(* PLC project TC3_TE1400_GeneratedModule_ModelBROSMattia_FB, Beckhoff Automation GmbH & Co. KG TwinCAT 3 Function - TE1400 1.2.1228 *)
(* stored: companyURL www.beckhoff.com, creationDateTime 2017-06-19T08:04:46 *)

TYPE E_TcMatSimDataAreaType : (NotSpecified := 0, Standard, InputSrc, InputDst, OutputSrc, OutputDst, InternalDa, MArea, RetainDa);
END_TYPE

TYPE ST_TcMatSimObjectDataAreaInfo : STRUCT
  pPlcVar : PVOID;
  pModuleProcImg : PVOID;
  nSize : UDINT;
  nDataAreaId : UDINT;
  eDataAreaType : E_TcMatSimDataAreaType;
END_STRUCT;
END_TYPE

{attribute 'pack_mode' := '4'}
TYPE ST_ModelBROSMattia_InitData : STRUCT
  Header : TComInitDataHdr;
  CallByHdr : TComInitDataElmHdr;
  CallBy : TctModuleCallByType;
  ExecutionSequenceHdr : TComInitDataElmHdr;
  ExecutionSequence : TctModuleExecutionSequenceType;
  StepSizeHdr : TComInitDataElmHdr;
  StepSize : TctStepSizeType;
  ExtendedFileAccessOIDHdr : TComInitDataElmHdr;
  ExtendedFileAccessOID : OTCID;
  ExtModeParametersHdr : TComInitDataElmHdr;
  ExtModeParameters : TctExtModeParametersType;
  ExecuteModelCodeHdr : TComInitDataElmHdr;
  ExecuteModelCode : BOOL;
  ModelParametersHdr : TComInitDataElmHdr;
  ModelParameters : P_model_bros_mattia_T;
  ContextInfoArr_0_TaskOidHdr : TComInitDataElmHdr;
  ContextInfoArr_0_TaskOid : OTCID;
  ContextInfoArr_0_TaskPriorityHdr : TComInitDataElmHdr;
  ContextInfoArr_0_TaskPriority : UDINT;
  ContextInfoArr_0_TaskCycleTimeNsHdr : TComInitDataElmHdr;
  ContextInfoArr_0_TaskCycleTimeNs : UDINT;
  ContextInfoArr_0_TaskPortHdr : TComInitDataElmHdr;
  ContextInfoArr_0_TaskPort : UINT;
  ContextInfoArr_0_TaskSortOrderHdr : TComInitDataElmHdr;
  ContextInfoArr_0_TaskSortOrder : UDINT;
END_STRUCT;
END_TYPE

TYPE ST_ModelBROSMattia_Input : STRUCT
  StatusWord_joint1 : UINT;
  MotorEncoder_joint1 : DINT;
  JointAbsEnc_joint1 : DINT;
  MotorCurrentAct_joint1 : INT;
  StatusWord_joint2 : UINT;
  MotorEncoder_joint2 : DINT;
  JointAbsEnc_joint2 : DINT;
  MotorCurrentAct_joint2 : INT;
  FTch1 : REAL;
  FTch2 : REAL;
  FTch3 : REAL;
  FTch4 : REAL;
  FTch5 : REAL;
  FTch6 : REAL;
  StatusWord_joint3 : UINT;
  MotorEncoder_joint3 : DINT;
  JointAbsEnc_joint3 : DINT;
  MotorCurrentAct_joint3 : INT;
  StatusWord_joint4 : UINT;
  MotorEncoder_joint4 : DINT;
  JointAbsEnc_joint4 : DINT;
  MotorCurrentAct_joint4 : INT;
  FTch7 : REAL;
  FTch8 : REAL;
  FTch9 : REAL;
  FTch10 : REAL;
  FTch11 : REAL;
  FTch12 : REAL;
END_STRUCT;
END_TYPE

TYPE ST_ModelBROSMattia_Output : STRUCT
  EnableCircuit1 : BOOL;
  ControlWord_joint1 : UINT;
  ModesOfOperation_joint1 : SINT;
  TargetCurrent_joint1 : INT;
  ControlWord_joint2 : UINT;
  ModesOfOperation_joint2 : SINT;
  TargetCurrent_joint2 : INT;
  EnableCircuit2 : BOOL;
  ControlWord_joint3 : UINT;
  ModesOfOperation_joint3 : SINT;
  TargetCurrent_joint3 : INT;
  ControlWord_joint4 : UINT;
  ModesOfOperation_joint4 : SINT;
  TargetCurrent_joint4 : INT;
  pause_logger : BOOL;
  DataToADS : matrix_9_real_T;
END_STRUCT;
END_TYPE

FUNCTION_BLOCK FB_TcMatSimObject
  VAR_INPUT
    bWriteFbInputValues : BOOL := TRUE;  (* set this flag to write FB input values to the TcComObject's input DataAreas. This will overwrite the mapped input values before module execution. Set to FALSE to read the mapped input values from the TcComObject to the FB. *)
  END_VAR
  VAR
    pDataAreas : POINTER TO ST_TcMatSimObjectDataAreaInfo;  (* process image src and dst pointers and sizes *)
    nDataAreas : UDINT;
    ipObjSrv : ITComObjectServer;  (* global interface pointers *)
    ipTcComObj : ITComObject;  (* object interface pointers *)
    ipTcCyclic : ITcCyclic;
    ipTcPostCyclic : ITcPostCyclic;
    ipTcAdi : ITcADI;
    ipTask : ITcTask;  (* task interface pointers *)
    pInitData : POINTER TO TComInitDataHdr;  (* initial parameters *)
    hResult : HRESULT;  (* hResult of interface calls (0 if no error) *)
    moduleClsId : CLSID;  (* module class ID *)
    assignedClsId : CLSID;  (* expected/desired module class ID *)
    bClassIdVerified : BOOL;
    bDynInstance : BOOL;  (* flag indicating whether the module instance was created dynamically *)
    eInitialObjState : TCOM_STATE := TCOM_STATE.TCOM_STATE_INIT;  (* the object state at the time FB_init was called, FB_exit will try to switch to this state (only if this means to shift down) *)
  END_VAR

            
          

{attribute 'object_name' := 'ReleaseTcComInterface'}
METHOD ReleaseTcComInterface : HRESULT
  VAR
    nStateChangeCnt : DINT := 0;
  END_VAR
                  
IF (ipTcComObj<>0) THEN
  WHILE (State>eInitialObjState AND nStateChangeCnt<1000) DO
    State := eInitialObjState;
    nStateChangeCnt := nStateChangeCnt+1;
  END_WHILE
  ReleaseObjInterfaces();
  IF (bDynInstance) THEN
    ReleaseTcComInterface := TC3_MODULE.FW_ObjMgr_DeleteInstance(ADR(ipTcComObj));
  ELSE
    ipTcComObj.TcRelease();
  END_IF
  ipTcComObj := 0;
END_IF
                  
                
END_METHOD

{attribute 'object_name' := 'ReleaseObjInterfaces'}
METHOD ReleaseObjInterfaces : HRESULT
                  
// release interface pointers
IF (ipTcCyclic<>0) THEN
  ipTcCyclic.TcRelease();
  ipTcCyclic := 0;
END_IF
IF (ipTcPostCyclic<>0) THEN
  ipTcPostCyclic.TcRelease();
  ipTcPostCyclic := 0;
END_IF
IF (ipTcAdi<>0) THEN
  ipTcAdi.TcRelease();
  ipTcAdi := 0;
END_IF
                  
                
END_METHOD

{attribute 'object_name' := 'Internal_SetObjState'}
METHOD Internal_SetObjState
  VAR_INPUT
    hr : REFERENCE TO HRESULT;
    nextState : TCOM_STATE;
  END_VAR
                  
// verify class id
IF (SUCCEEDED(hr)) THEN
  hr := VerifyClassId();
END_IF

// switch object state
IF (SUCCEEDED(hr) AND nextState>=TCOM_STATE_INIT) THEN
  IF (ipTcComObj=0) THEN
    hr := Tc2_System.E_HRESULTAdsErr.NOINTERFACE;
  END_IF
  IF (ipObjSrv=0) THEN
    hr := Tc2_System.E_HRESULTAdsErr.NOINTERFACE;
  END_IF
  IF (SUCCEEDED(hr)) THEN
    hr := ipTcComObj.TcSetObjState(nextState,ipObjSrv,pInitData);
  END_IF
END_IF
                  
                
END_METHOD

{attribute 'object_name' := 'FB_init'}
METHOD FB_init : BOOL
  VAR_INPUT
    bInitRetains : BOOL;  (* init retain variables *)
    bInCopyCode : BOOL;  (* Online Change *)
    oid : OTCID;
  END_VAR
                  
FB_init := SUCCEEDED(Init(oid));
                  
                
END_METHOD

{attribute 'object_name' := 'GetObjPara'}
METHOD GetObjPara : HRESULT
  VAR_INPUT
    pid : PTCID;
    nData : UDINT;
    pData : PVOID;
  END_VAR
                  
IF (ipTcComObj=0) THEN
  GetObjPara := Tc2_System.E_HRESULTAdsErr.NOINTERFACE;
END_IF

IF (SUCCEEDED(GetObjPara)) THEN
  GetObjPara := ipTcComObj.TcGetObjPara(pid:=pid,nData,pData,0);
END_IF
                  
                
END_METHOD

{attribute 'object_name' := 'QueryObjInterface'}
METHOD QueryObjInterface
  VAR_INPUT
    hr : REFERENCE TO HRESULT;
    iid : REFERENCE TO IID;
    pipItf : POINTER TO ITcUnknown;
  END_VAR
  VAR CONSTANT
    pNull : PVOID := 0;
  END_VAR
                  
IF (SUCCEEDED(hr)) THEN
  IF (ipTcComObj=0) THEN
    hr := Tc2_System.E_HRESULTAdsErr.NOINTERFACE;
  ELSIF (pipItf^=ULINT_TO_DWORD(pNull)) THEN
    hr := ipTcComObj.TcQueryInterface(iid:= iid, pipItf:=pipItf);
  END_IF
END_IF
                  
                
END_METHOD

{attribute 'object_name' := 'SaveOnlineParametersForInit'}
METHOD SaveOnlineParametersForInit : HRESULT
  VAR
    idx : UINT;
    pInitElemHdr : POINTER TO TComInitDataElmHdr;
    pData : PVOID;
    nData : UDINT;
  END_VAR
  VAR CONSTANT
    nInitDataAlignment : UDINT := 4;
  END_VAR
                  IF (pInitData<>0) THEN
  pInitElemHdr := pInitData + SIZEOF(pInitData^);
  FOR idx:=1 TO pInitData^.uiElmCnt DO
    pData := pInitElemHdr + ULINT_TO_DWORD(SIZEOF(pInitElemHdr^));
    nData := pInitElemHdr^.cbData;
    SaveOnlineParametersForInit := GetObjPara(pInitElemHdr^.indexOffset,nData,pData);
    IF (FAILED(SaveOnlineParametersForInit)) THEN
      RETURN;
    END_IF
    pInitElemHdr := pData + (nInitDataAlignment*((nData + nInitDataAlignment - 1)/nInitDataAlignment));
  END_FOR
ELSE
	SaveOnlineParametersForInit := Tc2_System.E_HRESULTAdsErr.NOTINIT;
END_IF
                  
                
END_METHOD

{attribute 'object_name' := 'ResetHresult'}
METHOD ResetHresult
                  hResult := S_OK;
                
END_METHOD

{attribute 'object_name' := 'Execute'}
METHOD Execute : HRESULT
  VAR
    nDaIdx : UDINT;
    pCurDataArea : POINTER TO ST_TcMatSimObjectDataAreaInfo;
  END_VAR
                  
IF (SUCCEEDED(hResult)) THEN
  hResult := VerifyClassId();
END_IF

IF (SUCCEEDED(hResult) AND State<>TCOM_STATE_OP) THEN
  hResult := Tc2_System.E_HRESULTAdsErr.NOTREADY;
END_IF

// get image pointers
IF (SUCCEEDED(hResult)) THEN
  GetImagePtrs(hResult);
END_IF

// copy inputs
IF (pDataAreas<>0 AND bWriteFbInputValues) THEN
  FOR nDaIdx:=0 TO nDataAreas-1 DO
    IF (FAILED(hResult))THEN
      CONTINUE;
    END_IF
    pCurDataArea := pDataAreas + nDaIdx*SIZEOF(ST_TcMatSimObjectDataAreaInfo);
    IF ((pCurDataArea^.eDataAreaType <> E_TcMatSimDataAreaType.InputDst))THEN
      CONTINUE;
    END_IF
    IF (pCurDataArea^.pModuleProcImg<>0 AND pCurDataArea^.pPlcVar<>0) THEN
      MEMCPY(pCurDataArea^.pModuleProcImg,pCurDataArea^.pPlcVar,pCurDataArea^.nSize);
    ELSE
      hResult := Tc2_System.E_HRESULTAdsErr.NOINTERFACE;
    END_IF
  END_FOR
END_IF

// call cycle update
IF (SUCCEEDED(hResult)) THEN
  IF (ipTcCyclic<>0) THEN
    hResult := ipTcCyclic.CycleUpdate(ipTask:= ipTask, ipCaller:= 0, context:= 0);
  ELSE
    hResult := Tc2_System.E_HRESULTAdsErr.NOINTERFACE;
  END_IF
END_IF

// copy outputs
IF (pDataAreas<>0) THEN
  FOR nDaIdx:=0 TO nDataAreas-1 DO
    IF (FAILED(hResult))THEN
      CONTINUE;
    END_IF
    pCurDataArea := pDataAreas + nDaIdx*SIZEOF(ST_TcMatSimObjectDataAreaInfo);
    IF ((pCurDataArea^.eDataAreaType = E_TcMatSimDataAreaType.OutputSrc) OR NOT bWriteFbInputValues) THEN
      IF (pCurDataArea^.pModuleProcImg<>0 AND pCurDataArea^.pPlcVar<>0) THEN
        MEMCPY(pCurDataArea^.pPlcVar,pCurDataArea^.pModuleProcImg,pCurDataArea^.nSize);
      ELSE
        hResult := Tc2_System.E_HRESULTAdsErr.NOINTERFACE;
      END_IF
    END_IF
  END_FOR
END_IF


// call post cyclic update
IF (SUCCEEDED(hResult)) THEN
  IF (ipTcPostCyclic<>0) THEN
    hResult := ipTcPostCyclic.PostCyclicUpdate(ipTask:= 0, ipCaller:= 0, context:= 0);
  ELSE
    hResult := Tc2_System.E_HRESULTAdsErr.NOINTERFACE;
  END_IF
END_IF

ReleaseImagePtrs();

Execute := hResult;
                  
                
END_METHOD

{attribute 'object_name' := 'GetImagePtrs'}
METHOD GetImagePtrs
  VAR_INPUT
    hr : REFERENCE TO HRESULT;
  END_VAR
  VAR
    nDaIdx : UDINT;
    pCurDataArea : POINTER TO ST_TcMatSimObjectDataAreaInfo;
  END_VAR
                  
IF (ipTcAdi=0) THEN
  hr := Tc2_System.E_HRESULTAdsErr.NOINTERFACE;
END_IF
IF(State<>TCOM_STATE_OP)THEN
  hr := Tc2_System.E_HRESULTAdsErr.INVALIDSTATE;
END_IF


// get pointers to process images
IF (pDataAreas<>0) THEN
  FOR nDaIdx:=0 TO nDataAreas-1 DO
    pCurDataArea := pDataAreas + nDaIdx*SIZEOF(ST_TcMatSimObjectDataAreaInfo);
    IF (FAILED(hr))THEN
      CONTINUE;
    END_IF
    IF ((pCurDataArea^.eDataAreaType <> E_TcMatSimDataAreaType.InputDst) AND (pCurDataArea^.eDataAreaType <> E_TcMatSimDataAreaType.OutputSrc))THEN
      CONTINUE;
    END_IF
    IF (pCurDataArea^.pModuleProcImg=0 AND pCurDataArea^.nSize>0) THEN
      hr := ipTcAdi.GetImagePtr(size:= pCurDataArea^.nSize , offs:=0 , adi_x:=pCurDataArea^.nDataAreaId , ppData:=ADR(pCurDataArea^.pModuleProcImg));
    END_IF
  END_FOR
END_IF

IF (FAILED(hr)) THEN
  ReleaseImagePtrs();
END_IF
                  
                
END_METHOD

{attribute 'object_name' := 'VerifyClassId'}
METHOD VerifyClassId : HRESULT
  VAR
    emptyClsId : CLSID;
  END_VAR
                  memset(ADR(emptyClsId),0,SIZEOF(emptyClsId));
IF (bClassIdVerified) THEN
  // class ID was already verified
  VerifyClassId := Tc2_System.E_HRESULTAdsErr.HRESULT_ADS_NOERROR;
ELSIF (memcmp(ADR(assignedClsId),ADR(emptyClsId),SIZEOF(assignedClsId))=0) THEN
  // skip class ID verification if no assignedClsId specified
  VerifyClassId := Tc2_System.E_HRESULTAdsErr.HRESULT_ADS_NOERROR;
ELSE
  // verify class ID
  VerifyClassId := ReadModuleClassId();

  IF (SUCCEEDED(VerifyClassId)) THEN
    IF (memcmp(ADR(assignedClsId),ADR(moduleClsId),SIZEOF(assignedClsId))<>0) THEN
     VerifyClassId := Tc2_System.E_HRESULTAdsErr.INVALIDCLSID;
    END_IF
  END_IF
  bClassIdVerified := SUCCEEDED(VerifyClassId);
END_IF
                  
                
END_METHOD

{attribute 'object_name' := 'SetObjPara'}
METHOD SetObjPara : HRESULT
  VAR_INPUT
    pid : PTCID;
    nData : UDINT;
    pData : PVOID;
  END_VAR
                  
IF (ipTcComObj=0) THEN
  SetObjPara := Tc2_System.E_HRESULTAdsErr.NOINTERFACE;
END_IF

IF (SUCCEEDED(SetObjPara)) THEN
  SetObjPara := ipTcComObj.TcSetObjPara(pid:=pid,nData,pData,0);
END_IF
                  
                
END_METHOD

{attribute 'object_name' := 'QueryTcComInterface'}
METHOD QueryTcComInterface
  VAR_INPUT
    hr : REFERENCE TO HRESULT;
    oid : OTCID;
  END_VAR
                  
IF (ipObjSrv=0) THEN
  hr := Tc2_System.E_HRESULTAdsErr.NOINTERFACE;
END_IF

IF (SUCCEEDED(hr) AND ipTcComObj=0) THEN
  bDynInstance := FALSE;
  IF(oid>0) THEN
    // query interface of existing object
    hr := ipObjSrv.TcQueryObjectInterface(oid,IID_ITComObject,ADR(ipTcComObj));
  ELSE
    // create new instance and get the object interface
    hr := ipObjSrv.TcCreateInstance(assignedClsId,IID_ITComObject,ADR(ipTcComObj));
    IF (SUCCEEDED(hr)) THEN
      bDynInstance := TRUE;
      hr := ipTcComObj.TcSetObjectId(OTCID_CreateNewId);
    END_IF
  END_IF
  IF (SUCCEEDED(hr)) THEN
    eInitialObjState := State;
  END_IF
END_IF
                  
                
END_METHOD

{attribute 'object_name' := 'ReleaseImagePtrs'}
METHOD ReleaseImagePtrs : HRESULT
  VAR
    nDaIdx : UDINT;
    pCurDataArea : POINTER TO ST_TcMatSimObjectDataAreaInfo;
  END_VAR
                  
IF (ipTcAdi=0) THEN
  ReleaseImagePtrs := Tc2_System.E_HRESULTAdsErr.NOINTERFACE;
END_IF

IF (SUCCEEDED(ReleaseImagePtrs) AND pDataAreas<>0) THEN
  // release pointers to the simulink module process images
  FOR nDaIdx:=0 TO nDataAreas-1 DO
    pCurDataArea := pDataAreas + nDaIdx*SIZEOF(ST_TcMatSimObjectDataAreaInfo);

    IF (pCurDataArea^.pModuleProcImg<>0) THEN
      ipTcAdi.ReleaseImagePtr(pData:=pCurDataArea^.pModuleProcImg);
      pCurDataArea^.pModuleProcImg := 0;
    END_IF
  END_FOR
END_IF
                  
                
END_METHOD

{attribute 'object_name' := 'FB_exit'}
METHOD FB_exit : BOOL
  VAR_INPUT
    bInCopyCode : BOOL;  (* Online Change *)
  END_VAR
                  
IF (NOT bInCopyCode) THEN
  IF (ipObjSrv<>0) THEN
    ipObjSrv.TcRelease();
    ipObjSrv := 0;
  END_IF

  ReleaseTcComInterface();
END_IF
                  
                
END_METHOD

{attribute 'object_name' := 'InitObjName'}
METHOD InitObjName
  VAR_INPUT
    hr : REFERENCE TO HRESULT;
  END_VAR
  VAR
    objectName : STRING(255) := 'TempContr_PlcRtFbInstance';
    oid : OTCID;
  END_VAR
                  
IF (SUCCEEDED(hr)) THEN
  hr := ipTcComObj.TcGetObjectId(oid);
END_IF

IF (SUCCEEDED(hr) and bDynInstance) THEN
  objectName := TC2_STANDARD.CONCAT(objectName,'_');
  objectName := TC2_STANDARD.CONCAT(objectName,UDINT_TO_STRING(oid));
  hr := ipTcComObj.TcSetObjectName(ADR(objectName));
END_IF
                  
                
END_METHOD

{attribute 'object_name' := 'SetObjState'}
METHOD SetObjState : HRESULT
  VAR_INPUT
    finalState : TCOM_STATE;
  END_VAR
  VAR
    bShiftUp : BOOL;
    bShiftDown : BOOL;
    currentState : TCOM_STATE;
  END_VAR
                  
currentState := State;

bShiftUp := finalState>currentState;
bShiftDown := finalState<currentState;

// do not switch up on error
IF (FAILED(hresult)) THEN
  bShiftUp := FALSE;
END_IF
// reset existing error on switching down
IF (bShiftDown) THEN
  ResetHresult();
END_IF

// prepared state switch
CASE currentState OF
  TCOM_STATE_INIT:
    IF(bShiftUp) THEN
      QueryTcComInterface(hResult,0);
      Internal_SetObjState(hResult,TCOM_STATE.TCOM_STATE_PREOP);
      InitObjName(hResult);
    END_IF

  TCOM_STATE_PREOP:
    IF(bShiftUp) THEN
      Internal_SetObjState(hResult,TCOM_STATE.TCOM_STATE_SAFEOP);
      QueryObjInterfaces(hResult);
    ELSIF (bShiftDown) THEN
      Internal_SetObjState(hResult,TCOM_STATE.TCOM_STATE_INIT);
    END_IF

  TCOM_STATE_SAFEOP:
    IF(bShiftUp) THEN
      Internal_SetObjState(hResult,TCOM_STATE.TCOM_STATE_OP);
      QueryObjInterfaces(hResult);
    ELSIF (bShiftDown) THEN
      Internal_SetObjState(hResult,TCOM_STATE.TCOM_STATE_PREOP);
      ReleaseObjInterfaces();
    END_IF


  TCOM_STATE_OP:
    IF (bShiftDown) THEN
      Internal_SetObjState(hResult,TCOM_STATE.TCOM_STATE_SAFEOP);
    END_IF
END_CASE

SetObjState := hResult;
                  
                
END_METHOD

{attribute 'object_name' := 'QueryObjInterfaces'}
METHOD QueryObjInterfaces
  VAR_INPUT
    hr : REFERENCE TO HRESULT;
  END_VAR
                  
IF(State<TCOM_STATE_PREOP)THEN
  hr := Tc2_System.E_HRESULTAdsErr.INVALIDSTATE;
END_IF

//cyclic interface
QueryObjInterface(hr,IID_ITCCYCLIC,ADR(ipTcCyclic));
//post cyclic interface
QueryObjInterface(hr,IID_ITCPOSTCYCLIC,ADR(ipTcPostCyclic));
//adi interface
QueryObjInterface(hr,IID_ITcADI,ADR(ipTcAdi));
                  
                
END_METHOD

{attribute 'object_name' := 'Init'}
METHOD Init : HRESULT
  VAR_INPUT
    oid : OTCID;
  END_VAR
                  
// preinitialize variables
memset(ADR(moduleClsId),0,SIZEOF(moduleClsId));
bClassIdVerified := FALSE;
hResult := Tc2_System.E_HRESULTAdsErr.HRESULT_ADS_NOERROR;

// get object server
IF (ipObjSrv=0) THEN
  hResult := FW_ObjMgr_GetObjectServer(_AppInfo.ObjId,ADR(ipObjSrv));
END_IF

// try to get object interfaces
IF (SUCCEEDED(hresult)) THEN
  QueryTcComInterface(hResult,oid);
END_IF

// verify class id
IF (SUCCEEDED(hresult)) THEN
  hresult := VerifyClassId();
END_IF

// query interfaces, if the current state is higher than INIT
IF (SUCCEEDED(hresult) AND State>TCOM_STATE.TCOM_STATE_INIT) THEN
  QueryObjInterfaces(hResult);
END_IF

// return value
Init := hresult;
                  
                
END_METHOD

{attribute 'object_name' := 'ReadModuleClassId'}
METHOD ReadModuleClassId : HRESULT
  VAR
    emptyClsId : CLSID;
  END_VAR
                  memset(ADR(emptyClsId),0,SIZEOF(emptyClsId));
IF (memcmp(ADR(moduleClsId),ADR(emptyClsId),SIZEOF(moduleClsId))=0) THEN
  IF (ipTcComObj=0) THEN
    ReadModuleClassId := Tc2_System.E_HRESULTAdsErr.NOINTERFACE;
  END_IF

  //objectClsId := clsid;
  IF (SUCCEEDED(ReadModuleClassId)) THEN
    ReadModuleClassId := ipTcComObj.GetClassId(moduleClsId);
  END_IF
END_IF
                
END_METHOD

METHOD PUBLIC AssignClassId
VAR_INPUT
	clsId : CLSID;
END_VAR
                  assignedClsId := clsId;
bClassIdVerified := false;
                  
                
END_METHOD

PROPERTY Error : BOOL
GET
                    Error := FAILED(hResult);
                  
END_GET
END_PROPERTY

METHOD PUBLIC SetDataAreaInfo
VAR_INPUT
  pDataAreas: POINTER TO ST_TcMatSimObjectDataAreaInfo;
  nDataAreas: UDINT;
END_VAR
                  
THIS^.nDataAreas := nDataAreas;
THIS^.pDataAreas := pDataAreas;
                  
                
END_METHOD

METHOD PUBLIC SetInitDataInfo
VAR_INPUT
  pInitData : POINTER TO TComInitDataHdr;
END_VAR
                  this^.pInitData := pInitData;
                
END_METHOD

PROPERTY ClassId : CLSID
GET
                    hResult := ReadModuleClassId();
ClassId := moduleClsId;
                    
                  
END_GET
END_PROPERTY

PROPERTY State : TCOM_STATE
GET
  VAR
    hr : HRESULT := S_OK;
    eObjState : TCOM_STATE;
  END_VAR
                    
IF (ipTcComObj<>0) THEN
  hr := ipTcComObj.TcGetObjState(ADR(eObjState));
IF (FAILED(hr)) THEN
  eObjState := TCOM_STATE.TCOM_STATE_INIT;
END_IF
ELSE
  eObjState := TCOM_STATE.TCOM_STATE_INIT;
END_IF
State := eObjState;
                    
                  
END_GET
SET
                    SetObjState(State);
                  
END_SET
END_PROPERTY

PROPERTY ErrorCode : HRESULT
GET
                    ErrorCode := hResult;
                  
END_GET
END_PROPERTY
END_FUNCTION_BLOCK

{attribute 'TcDependOnClassFactory' := 'ModelBROSMattia'}
FUNCTION_BLOCK FB_ModelBROSMattia EXTENDS FB_TcMatSimObject
  VAR_INPUT
    stInput : ST_ModelBROSMattia_Input;
  END_VAR
  VAR_OUTPUT
    stOutput : ST_ModelBROSMattia_Output;
  END_VAR
  VAR
    stInitData : ST_ModelBROSMattia_InitData;
    arrDataAreas : ARRAY[1..2] OF ST_TcMatSimObjectDataAreaInfo;
    bParametersVerified : BOOL;
  END_VAR

            
          

{attribute 'object_name' := 'Internal_SetObjState'}
METHOD Internal_SetObjState
  VAR_INPUT
    hr : REFERENCE TO HRESULT;
    nextState : TCOM_STATE;
  END_VAR
                  
// update pointer to InitData structure
SetInitDataInfo(ADR(stInitData));
// call base method
SUPER^.Internal_SetObjState(hr,nextState);
                  
                
END_METHOD

{attribute 'object_name' := 'SaveOnlineParametersForInit'}
METHOD SaveOnlineParametersForInit : HRESULT
  VAR
    idx : UINT;
    pInitElemHdr : POINTER TO TComInitDataElmHdr;
    pData : PVOID;
    nData : UDINT;
  END_VAR
  VAR CONSTANT
    nInitDataAlignment : UDINT := 4;
  END_VAR
                  
// update pointer to InitData structure
SetInitDataInfo(ADR(stInitData));
// call base method
SaveOnlineParametersForInit := SUPER^.SaveOnlineParametersForInit();
                  
                
END_METHOD

METHOD FB_init : BOOL
  VAR_INPUT
    bInitRetains : BOOL;  (* if TRUE, the retain variables are initialized (warm start / cold start) *)
    bInCopyCode : BOOL;  (* if TRUE, the instance afterwards gets moved into the copy code (online change) *)
    oid : OTCID;
  END_VAR
  VAR
    clsId : CLSID;
  END_VAR
                  
// initialize flags
bParametersVerified := false;
                    
// set module class id for compatibility check
clsId.Data1 := 16#e004bc57;
clsId.Data2 := 16#472f;
clsId.Data3 := 16#4bf7;
clsId.Data4[0] := 16#85;
clsId.Data4[1] := 16#bd;
clsId.Data4[2] := 16#47;
clsId.Data4[3] := 16#db;
clsId.Data4[4] := 16#44;
clsId.Data4[5] := 16#05;
clsId.Data4[6] := 16#27;
clsId.Data4[7] := 16#ce;

AssignClassId(clsId);
                    
// initialize InitData structure with default values              
stInitData.CallByHdr.indexGroup := 0;
stInitData.CallByHdr.indexOffset := 16#00000000;
stInitData.CallByHdr.cbData := SIZEOF(stInitData.CallBy);
stInitData.CallBy := TctModuleCallByType.CyclicTask;
stInitData.ExecutionSequenceHdr.indexGroup := 0;
stInitData.ExecutionSequenceHdr.indexOffset := 16#00000001;
stInitData.ExecutionSequenceHdr.cbData := SIZEOF(stInitData.ExecutionSequence);
stInitData.ExecutionSequence := TctModuleExecutionSequenceType.StateUpdateAfterOutputMapping;
stInitData.StepSizeHdr.indexGroup := 0;
stInitData.StepSizeHdr.indexOffset := 16#00000002;
stInitData.StepSizeHdr.cbData := SIZEOF(stInitData.StepSize);
stInitData.StepSize := TctStepSizeType.RequireMatchingTaskCycleTime;
stInitData.ExtendedFileAccessOIDHdr.indexGroup := 0;
stInitData.ExtendedFileAccessOIDHdr.indexOffset := 16#00000005;
stInitData.ExtendedFileAccessOIDHdr.cbData := SIZEOF(stInitData.ExtendedFileAccessOID);
stInitData.ExtendedFileAccessOID := 0;
stInitData.ExtModeParametersHdr.indexGroup := 0;
stInitData.ExtModeParametersHdr.indexOffset := 16#bf002000;
stInitData.ExtModeParametersHdr.cbData := SIZEOF(stInitData.ExtModeParameters);
stInitData.ExtModeParameters.ConnectionTimeout := 3;
stInitData.ExtModeParameters.InitIncomingPktBufferSize := 10000;
stInitData.ExtModeParameters.InitOutgoingPktBufferSize := 10000;
stInitData.ExtModeParameters.Activated := 1;
stInitData.ExtModeParameters.AllowExecutionCommands := 1;
stInitData.ExtModeParameters.WaitForStartCommand := 0;
stInitData.ExtModeParameters.AllowParameterChange := 1;
stInitData.ExecuteModelCodeHdr.indexGroup := 0;
stInitData.ExecuteModelCodeHdr.indexOffset := 16#00000008;
stInitData.ExecuteModelCodeHdr.cbData := SIZEOF(stInitData.ExecuteModelCode);
stInitData.ExecuteModelCode := 1;
stInitData.ModelParametersHdr.indexGroup := 0;
stInitData.ModelParametersHdr.indexOffset := 16#83000000;
stInitData.ModelParametersHdr.cbData := SIZEOF(stInitData.ModelParameters);
stInitData.ModelParameters.FM1.HomeLocationOpSpace[0] := 0;
stInitData.ModelParameters.FM1.HomeLocationOpSpace[1] := 0.25;
stInitData.ModelParameters.FM1.HomeLocationSize := 0.0025;
stInitData.ModelParameters.FM1.NominalPositionOpSpace[0] := 0;
stInitData.ModelParameters.FM1.NominalPositionOpSpace[1] := 0.25;
stInitData.ModelParameters.FM1.DynModParams[0] := 0.0009446018;
stInitData.ModelParameters.FM1.DynModParams[1] := 0.0005536255;
stInitData.ModelParameters.FM1.DynModParams[2] := 0.1102026;
stInitData.ModelParameters.FM1.DynModParams[3] := 0.1175426;
stInitData.ModelParameters.FM1.DynModParams[4] := -0.006234047;
stInitData.ModelParameters.FM1.DynModParams[5] := 0.1037213;
stInitData.ModelParameters.FM1.DynModParams[6] := 0.003853734;
stInitData.ModelParameters.FM1.Actuator1.JointAbsoluteEncoderCounts_rev := 65536;
stInitData.ModelParameters.FM1.Actuator1.AbsEncoderOffset := 5.303223547422882;
stInitData.ModelParameters.FM1.Actuator1.MotorEncoderCounts_rev := 4096;
stInitData.ModelParameters.FM1.Actuator1.FOAWNoiseLevel := 0.0009;
stInitData.ModelParameters.FM1.Actuator1.transmissionRatio := 7.2976;
stInitData.ModelParameters.FM1.Actuator1.motorTorqueConstant := 0.08486;
stInitData.ModelParameters.FM1.Actuator1.drivePeakCurrent := 20;
stInitData.ModelParameters.FM1.Actuator1.AbsoluteMaximumTorque_Nm := 8;
stInitData.ModelParameters.FM1.Actuator1.TransmissionSlipAngleGuardMax := 0.08726646259971647;
stInitData.ModelParameters.FM1.Actuator1.JointPositionGuardMin := -0.4363323129985824;
stInitData.ModelParameters.FM1.Actuator1.JointPositionGuardMax := 2.356194490192345;
stInitData.ModelParameters.FM1.Actuator1.FilterButterA[0] := 1;
stInitData.ModelParameters.FM1.Actuator1.FilterButterA[1] := -1.475480443592646;
stInitData.ModelParameters.FM1.Actuator1.FilterButterA[2] := 0.5869195080611904;
stInitData.ModelParameters.FM1.Actuator1.FilterButterB[0] := 0.02785976611713603;
stInitData.ModelParameters.FM1.Actuator1.FilterButterB[1] := 0.05571953223427206;
stInitData.ModelParameters.FM1.Actuator1.FilterButterB[2] := 0.02785976611713603;
stInitData.ModelParameters.FM1.Actuator2.JointAbsoluteEncoderCounts_rev := 65536;
stInitData.ModelParameters.FM1.Actuator2.AbsEncoderOffset := 7.340133727728301;
stInitData.ModelParameters.FM1.Actuator2.MotorEncoderCounts_rev := 4096;
stInitData.ModelParameters.FM1.Actuator2.FOAWNoiseLevel := 0.0009;
stInitData.ModelParameters.FM1.Actuator2.transmissionRatio := 7.331;
stInitData.ModelParameters.FM1.Actuator2.motorTorqueConstant := 0.08486;
stInitData.ModelParameters.FM1.Actuator2.drivePeakCurrent := 20;
stInitData.ModelParameters.FM1.Actuator2.AbsoluteMaximumTorque_Nm := 8;
stInitData.ModelParameters.FM1.Actuator2.TransmissionSlipAngleGuardMax := 0.08726646259971647;
stInitData.ModelParameters.FM1.Actuator2.JointPositionGuardMin := 0.7853981633974483;
stInitData.ModelParameters.FM1.Actuator2.JointPositionGuardMax := 3.577924966588375;
stInitData.ModelParameters.FM1.Actuator2.FilterButterA[0] := 1;
stInitData.ModelParameters.FM1.Actuator2.FilterButterA[1] := -1.475480443592646;
stInitData.ModelParameters.FM1.Actuator2.FilterButterA[2] := 0.5869195080611904;
stInitData.ModelParameters.FM1.Actuator2.FilterButterB[0] := 0.02785976611713603;
stInitData.ModelParameters.FM1.Actuator2.FilterButterB[1] := 0.05571953223427206;
stInitData.ModelParameters.FM1.Actuator2.FilterButterB[2] := 0.02785976611713603;
stInitData.ModelParameters.FM1.FTSensor.MaxAllowableForcesTorqueSensor[0] := 70;
stInitData.ModelParameters.FM1.FTSensor.MaxAllowableForcesTorqueSensor[1] := 70;
stInitData.ModelParameters.FM1.FTSensor.MaxAllowableForcesTorqueSensor[2] := 140;
stInitData.ModelParameters.FM1.FTSensor.MaxAllowableForcesTorqueSensor[3] := 1.4;
stInitData.ModelParameters.FM1.FTSensor.MaxAllowableForcesTorqueSensor[4] := 1.4;
stInitData.ModelParameters.FM1.FTSensor.MaxAllowableForcesTorqueSensor[5] := 1.4;
stInitData.ModelParameters.FM1.FTSensor.TransformationMatrixSide := 1;
stInitData.ModelParameters.FM2.HomeLocationOpSpace[0] := 0;
stInitData.ModelParameters.FM2.HomeLocationOpSpace[1] := 0.25;
stInitData.ModelParameters.FM2.HomeLocationSize := 0.0025;
stInitData.ModelParameters.FM2.NominalPositionOpSpace[0] := 0;
stInitData.ModelParameters.FM2.NominalPositionOpSpace[1] := 0.25;
stInitData.ModelParameters.FM2.DynModParams[0] := 0.001117256;
stInitData.ModelParameters.FM2.DynModParams[1] := 0.0012246;
stInitData.ModelParameters.FM2.DynModParams[2] := 0.08800769;
stInitData.ModelParameters.FM2.DynModParams[3] := 0.1073326;
stInitData.ModelParameters.FM2.DynModParams[4] := 0.001462254;
stInitData.ModelParameters.FM2.DynModParams[5] := 0.1416925;
stInitData.ModelParameters.FM2.DynModParams[6] := 0.006135432;
stInitData.ModelParameters.FM2.Actuator1.JointAbsoluteEncoderCounts_rev := 65536;
stInitData.ModelParameters.FM2.Actuator1.AbsEncoderOffset := 3.23580094055001;
stInitData.ModelParameters.FM2.Actuator1.MotorEncoderCounts_rev := 4096;
stInitData.ModelParameters.FM2.Actuator1.FOAWNoiseLevel := 0.0009;
stInitData.ModelParameters.FM2.Actuator1.transmissionRatio := 7.3607;
stInitData.ModelParameters.FM2.Actuator1.motorTorqueConstant := 0.08486;
stInitData.ModelParameters.FM2.Actuator1.drivePeakCurrent := 20;
stInitData.ModelParameters.FM2.Actuator1.AbsoluteMaximumTorque_Nm := 8;
stInitData.ModelParameters.FM2.Actuator1.TransmissionSlipAngleGuardMax := 0.08726646259971647;
stInitData.ModelParameters.FM2.Actuator1.JointPositionGuardMin := -0.4363323129985824;
stInitData.ModelParameters.FM2.Actuator1.JointPositionGuardMax := 2.356194490192345;
stInitData.ModelParameters.FM2.Actuator1.FilterButterA[0] := 1;
stInitData.ModelParameters.FM2.Actuator1.FilterButterA[1] := -1.475480443592646;
stInitData.ModelParameters.FM2.Actuator1.FilterButterA[2] := 0.5869195080611904;
stInitData.ModelParameters.FM2.Actuator1.FilterButterB[0] := 0.02785976611713603;
stInitData.ModelParameters.FM2.Actuator1.FilterButterB[1] := 0.05571953223427206;
stInitData.ModelParameters.FM2.Actuator1.FilterButterB[2] := 0.02785976611713603;
stInitData.ModelParameters.FM2.Actuator2.JointAbsoluteEncoderCounts_rev := 65536;
stInitData.ModelParameters.FM2.Actuator2.AbsEncoderOffset := 4.445224359590367;
stInitData.ModelParameters.FM2.Actuator2.MotorEncoderCounts_rev := 4096;
stInitData.ModelParameters.FM2.Actuator2.FOAWNoiseLevel := 0.0009;
stInitData.ModelParameters.FM2.Actuator2.transmissionRatio := 7.32214;
stInitData.ModelParameters.FM2.Actuator2.motorTorqueConstant := 0.08486;
stInitData.ModelParameters.FM2.Actuator2.drivePeakCurrent := 20;
stInitData.ModelParameters.FM2.Actuator2.AbsoluteMaximumTorque_Nm := 8;
stInitData.ModelParameters.FM2.Actuator2.TransmissionSlipAngleGuardMax := 0.08726646259971647;
stInitData.ModelParameters.FM2.Actuator2.JointPositionGuardMin := 0.7853981633974483;
stInitData.ModelParameters.FM2.Actuator2.JointPositionGuardMax := 3.577924966588375;
stInitData.ModelParameters.FM2.Actuator2.FilterButterA[0] := 1;
stInitData.ModelParameters.FM2.Actuator2.FilterButterA[1] := -1.475480443592646;
stInitData.ModelParameters.FM2.Actuator2.FilterButterA[2] := 0.5869195080611904;
stInitData.ModelParameters.FM2.Actuator2.FilterButterB[0] := 0.02785976611713603;
stInitData.ModelParameters.FM2.Actuator2.FilterButterB[1] := 0.05571953223427206;
stInitData.ModelParameters.FM2.Actuator2.FilterButterB[2] := 0.02785976611713603;
stInitData.ModelParameters.FM2.FTSensor.MaxAllowableForcesTorqueSensor[0] := 70;
stInitData.ModelParameters.FM2.FTSensor.MaxAllowableForcesTorqueSensor[1] := 70;
stInitData.ModelParameters.FM2.FTSensor.MaxAllowableForcesTorqueSensor[2] := 140;
stInitData.ModelParameters.FM2.FTSensor.MaxAllowableForcesTorqueSensor[3] := 1.4;
stInitData.ModelParameters.FM2.FTSensor.MaxAllowableForcesTorqueSensor[4] := 1.4;
stInitData.ModelParameters.FM2.FTSensor.MaxAllowableForcesTorqueSensor[5] := 1.4;
stInitData.ModelParameters.FM2.FTSensor.TransformationMatrixSide := 2;
stInitData.ModelParameters.Ax_filt[0] := 0.964232663461483;
stInitData.ModelParameters.Ax_filt[1] := 0.9180119591620001;
stInitData.ModelParameters.Ax_filt[2] := 0.8316962937356224;
stInitData.ModelParameters.Ax_filt[3] := 0.6861219507280224;
stInitData.ModelParameters.Ax_filt[4] := 0.5095551888664519;
stInitData.ModelParameters.Ax_filt[5] := 0.3747475061520537;
stInitData.ModelParameters.Ay_filt[0] := 0.9540282163784651;
stInitData.ModelParameters.Ay_filt[1] := 0.8906519727779925;
stInitData.ModelParameters.Ay_filt[2] := 0.8014870484078772;
stInitData.ModelParameters.Ay_filt[3] := 0.6598213090970109;
stInitData.ModelParameters.Ay_filt[4] := 0.5276098539016424;
stInitData.ModelParameters.Ay_filt[5] := 0.3552761669082853;
stInitData.ModelParameters.Lb := 0.07000000000000001;
stInitData.ModelParameters.Lf := 0.238;
stInitData.ModelParameters.Lu := 0.153;
stInitData.ModelParameters.max_radius_target := 0.08;
stInitData.ModelParameters.maxofx_target[0] := 3.374735080502004;
stInitData.ModelParameters.maxofx_target[1] := 3.279975107067715;
stInitData.ModelParameters.maxofx_target[2] := 3.178225721986778;
stInitData.ModelParameters.maxofx_target[3] := 3.39423651654402;
stInitData.ModelParameters.maxofx_target[4] := 3.150914535434884;
stInitData.ModelParameters.maxofx_target[5] := 3.350920975347514;
stInitData.ModelParameters.maxofx_target[6] := 2.991162345696621;
stInitData.ModelParameters.maxofx_target[7] := 3.078293077059009;
stInitData.ModelParameters.maxofx_target[8] := 3.0526194754007;
stInitData.ModelParameters.maxofx_target[9] := 3.174093635233409;
stInitData.ModelParameters.maxofx_target[10] := 3.156570764399686;
stInitData.ModelParameters.maxofx_target[11] := 3.369201892278452;
stInitData.ModelParameters.maxofx_target[12] := 3.114402551583243;
stInitData.ModelParameters.maxofx_target[13] := 2.918380662381565;
stInitData.ModelParameters.maxofx_target[14] := 3.143318713585403;
stInitData.ModelParameters.maxofx_target[15] := 3.122666815693063;
stInitData.ModelParameters.maxofx_target[16] := 3.052430398243802;
stInitData.ModelParameters.maxofx_target[17] := 3.252001001363745;
stInitData.ModelParameters.maxofx_target[18] := 3.343115538099071;
stInitData.ModelParameters.maxofx_target[19] := 3.073425174954439;
stInitData.ModelParameters.maxofy_target[0] := 3.149069528347376;
stInitData.ModelParameters.maxofy_target[1] := 3.231961318092376;
stInitData.ModelParameters.maxofy_target[2] := 3.099601450389282;
stInitData.ModelParameters.maxofy_target[3] := 3.26658102122961;
stInitData.ModelParameters.maxofy_target[4] := 3.332313324019208;
stInitData.ModelParameters.maxofy_target[5] := 3.281602907608862;
stInitData.ModelParameters.maxofy_target[6] := 3.013770389116802;
stInitData.ModelParameters.maxofy_target[7] := 3.228221719839184;
stInitData.ModelParameters.maxofy_target[8] := 3.108979119108026;
stInitData.ModelParameters.maxofy_target[9] := 3.53401236222931;
stInitData.ModelParameters.maxofy_target[10] := 3.143674810712946;
stInitData.ModelParameters.maxofy_target[11] := 3.13643716203597;
stInitData.ModelParameters.maxofy_target[12] := 3.50914004294165;
stInitData.ModelParameters.maxofy_target[13] := 3.304014737714594;
stInitData.ModelParameters.maxofy_target[14] := 3.203259781107545;
stInitData.ModelParameters.maxofy_target[15] := 3.359348245482384;
stInitData.ModelParameters.maxofy_target[16] := 3.319663333123807;
stInitData.ModelParameters.maxofy_target[17] := 3.117503369285954;
stInitData.ModelParameters.maxofy_target[18] := 3.263182983320035;
stInitData.ModelParameters.maxofy_target[19] := 3.095487175408008;
stInitData.ModelParameters.nx_target[0] := 7;
stInitData.ModelParameters.nx_target[1] := 11;
stInitData.ModelParameters.nx_target[2] := 17;
stInitData.ModelParameters.nx_target[3] := 27;
stInitData.ModelParameters.nx_target[4] := 43;
stInitData.ModelParameters.nx_target[5] := 63;
stInitData.ModelParameters.ny_target[0] := 8;
stInitData.ModelParameters.ny_target[1] := 13;
stInitData.ModelParameters.ny_target[2] := 19;
stInitData.ModelParameters.ny_target[3] := 29;
stInitData.ModelParameters.ny_target[4] := 41;
stInitData.ModelParameters.ny_target[5] := 67;
stInitData.ModelParameters.phasesx_target[0] := 1.054129575369354;
stInitData.ModelParameters.phasesx_target[1] := -8.984668868752456;
stInitData.ModelParameters.phasesx_target[2] := 4.684012620994619;
stInitData.ModelParameters.phasesx_target[3] := -1.78041163347793;
stInitData.ModelParameters.phasesx_target[4] := 12.33404044654894;
stInitData.ModelParameters.phasesx_target[5] := -8.493502170828631;
stInitData.ModelParameters.phasesx_target[6] := -12.69343558803834;
stInitData.ModelParameters.phasesx_target[7] := -4.328255166789693;
stInitData.ModelParameters.phasesx_target[8] := -0.2154929352791773;
stInitData.ModelParameters.phasesx_target[9] := 5.448826103659846;
stInitData.ModelParameters.phasesx_target[10] := 6.369843261974847;
stInitData.ModelParameters.phasesx_target[11] := -0.9688373669540356;
stInitData.ModelParameters.phasesx_target[12] := -3.725435918561739;
stInitData.ModelParameters.phasesx_target[13] := -7.608070244880908;
stInitData.ModelParameters.phasesx_target[14] := 6.774707882496031;
stInitData.ModelParameters.phasesx_target[15] := 11.35903106494959;
stInitData.ModelParameters.phasesx_target[16] := 8.939459044730215;
stInitData.ModelParameters.phasesx_target[17] := 3.3240695074699;
stInitData.ModelParameters.phasesx_target[18] := 5.651857033576386;
stInitData.ModelParameters.phasesx_target[19] := 5.660625389351311;
stInitData.ModelParameters.phasesx_target[20] := 6.052043447445772;
stInitData.ModelParameters.phasesx_target[21] := 0.1123381420814134;
stInitData.ModelParameters.phasesx_target[22] := -7.691393321586861;
stInitData.ModelParameters.phasesx_target[23] := -5.658666496600078;
stInitData.ModelParameters.phasesx_target[24] := 7.822687631883769;
stInitData.ModelParameters.phasesx_target[25] := 9.875291825680804;
stInitData.ModelParameters.phasesx_target[26] := -10.13827695401784;
stInitData.ModelParameters.phasesx_target[27] := -9.07065425599488;
stInitData.ModelParameters.phasesx_target[28] := -13.83589092817621;
stInitData.ModelParameters.phasesx_target[29] := -2.336179842402662;
stInitData.ModelParameters.phasesx_target[30] := 0.02671956952722981;
stInitData.ModelParameters.phasesx_target[31] := 0.3557775666008609;
stInitData.ModelParameters.phasesx_target[32] := -4.374349654841463;
stInitData.ModelParameters.phasesx_target[33] := 8.476109776386904;
stInitData.ModelParameters.phasesx_target[34] := -15.32933899106938;
stInitData.ModelParameters.phasesx_target[35] := 6.772193739169005;
stInitData.ModelParameters.phasesx_target[36] := 7.375983992915446;
stInitData.ModelParameters.phasesx_target[37] := -2.728589976436413;
stInitData.ModelParameters.phasesx_target[38] := 4.523518253684084;
stInitData.ModelParameters.phasesx_target[39] := -1.980190294220159;
stInitData.ModelParameters.phasesx_target[40] := -11.72891380690488;
stInitData.ModelParameters.phasesx_target[41] := -1.616905542112287;
stInitData.ModelParameters.phasesx_target[42] := 3.843505538968176;
stInitData.ModelParameters.phasesx_target[43] := -5.776984566529401;
stInitData.ModelParameters.phasesx_target[44] := -6.535128534661852;
stInitData.ModelParameters.phasesx_target[45] := -0.9603240416738175;
stInitData.ModelParameters.phasesx_target[46] := -4.293274840505548;
stInitData.ModelParameters.phasesx_target[47] := 8.107261392713681;
stInitData.ModelParameters.phasesx_target[48] := -8.5268379035588;
stInitData.ModelParameters.phasesx_target[49] := 0.3063040941215773;
stInitData.ModelParameters.phasesx_target[50] := 17.68591556650787;
stInitData.ModelParameters.phasesx_target[51] := -1.186586826238688;
stInitData.ModelParameters.phasesx_target[52] := 1.488294868508662;
stInitData.ModelParameters.phasesx_target[53] := -1.587630120792048;
stInitData.ModelParameters.phasesx_target[54] := -6.350312023229334;
stInitData.ModelParameters.phasesx_target[55] := 4.230280867000283;
stInitData.ModelParameters.phasesx_target[56] := -3.683811749041483;
stInitData.ModelParameters.phasesx_target[57] := -6.980914393783903;
stInitData.ModelParameters.phasesx_target[58] := 3.772432609592454;
stInitData.ModelParameters.phasesx_target[59] := -7.676766307898628;
stInitData.ModelParameters.phasesx_target[60] := -8.963344830289831;
stInitData.ModelParameters.phasesx_target[61] := -7.290937359334666;
stInitData.ModelParameters.phasesx_target[62] := 1.53172869077159;
stInitData.ModelParameters.phasesx_target[63] := -4.21075624526638;
stInitData.ModelParameters.phasesx_target[64] := 5.838201626927779;
stInitData.ModelParameters.phasesx_target[65] := 3.067679012844269;
stInitData.ModelParameters.phasesx_target[66] := -6.782599631837804;
stInitData.ModelParameters.phasesx_target[67] := 11.67260587271691;
stInitData.ModelParameters.phasesx_target[68] := -1.369744477791799;
stInitData.ModelParameters.phasesx_target[69] := -9.769727430294244;
stInitData.ModelParameters.phasesx_target[70] := -1.03801189603194;
stInitData.ModelParameters.phasesx_target[71] := 3.934463295442507;
stInitData.ModelParameters.phasesx_target[72] := -6.303952092087981;
stInitData.ModelParameters.phasesx_target[73] := -8.814569770278936;
stInitData.ModelParameters.phasesx_target[74] := 1.332979314892913;
stInitData.ModelParameters.phasesx_target[75] := -2.930537832331445;
stInitData.ModelParameters.phasesx_target[76] := -7.199237600290243;
stInitData.ModelParameters.phasesx_target[77] := -4.636462839747684;
stInitData.ModelParameters.phasesx_target[78] := 4.656664603417048;
stInitData.ModelParameters.phasesx_target[79] := -2.453589570819968;
stInitData.ModelParameters.phasesx_target[80] := -6.648204718177245;
stInitData.ModelParameters.phasesx_target[81] := 1.916674251395496;
stInitData.ModelParameters.phasesx_target[82] := 14.59321971249467;
stInitData.ModelParameters.phasesx_target[83] := 2.233246872287854;
stInitData.ModelParameters.phasesx_target[84] := 2.552858747285482;
stInitData.ModelParameters.phasesx_target[85] := 1.636380635245875;
stInitData.ModelParameters.phasesx_target[86] := -3.476916590986135;
stInitData.ModelParameters.phasesx_target[87] := 3.877253330517075;
stInitData.ModelParameters.phasesx_target[88] := 2.65668364275337;
stInitData.ModelParameters.phasesx_target[89] := -9.996015286747692;
stInitData.ModelParameters.phasesx_target[90] := 4.283869437272529;
stInitData.ModelParameters.phasesx_target[91] := 1.488007350762337;
stInitData.ModelParameters.phasesx_target[92] := 3.554771691388678;
stInitData.ModelParameters.phasesx_target[93] := -7.262897562007865;
stInitData.ModelParameters.phasesx_target[94] := -2.820275901847407;
stInitData.ModelParameters.phasesx_target[95] := 1.715745541188431;
stInitData.ModelParameters.phasesx_target[96] := -5.91917503601243;
stInitData.ModelParameters.phasesx_target[97] := -8.098337380579832;
stInitData.ModelParameters.phasesx_target[98] := 4.374745632992884;
stInitData.ModelParameters.phasesx_target[99] := -7.504594463087322;
stInitData.ModelParameters.phasesx_target[100] := -1.004665776811523;
stInitData.ModelParameters.phasesx_target[101] := 5.372086109655486;
stInitData.ModelParameters.phasesx_target[102] := -2.000364289817965;
stInitData.ModelParameters.phasesx_target[103] := 5.625708687849259;
stInitData.ModelParameters.phasesx_target[104] := -3.604733381777346;
stInitData.ModelParameters.phasesx_target[105] := 9.163468645447979;
stInitData.ModelParameters.phasesx_target[106] := 9.569784090304315;
stInitData.ModelParameters.phasesx_target[107] := -9.983579856163516;
stInitData.ModelParameters.phasesx_target[108] := 0.6506750236191189;
stInitData.ModelParameters.phasesx_target[109] := -14.84719359184144;
stInitData.ModelParameters.phasesx_target[110] := 11.17211140642172;
stInitData.ModelParameters.phasesx_target[111] := -3.247697138772289;
stInitData.ModelParameters.phasesx_target[112] := -3.078275512995333;
stInitData.ModelParameters.phasesx_target[113] := -10.30653736918848;
stInitData.ModelParameters.phasesx_target[114] := -11.82059025223983;
stInitData.ModelParameters.phasesx_target[115] := 2.497529028681385;
stInitData.ModelParameters.phasesx_target[116] := 7.039003684349792;
stInitData.ModelParameters.phasesx_target[117] := 7.036957557540296;
stInitData.ModelParameters.phasesx_target[118] := -4.218399305616489;
stInitData.ModelParameters.phasesx_target[119] := 3.298395085669102;
stInitData.ModelParameters.phasesy_target[0] := -7.600292490432392;
stInitData.ModelParameters.phasesy_target[1] := -4.575825387822675;
stInitData.ModelParameters.phasesy_target[2] := 0.572202617583946;
stInitData.ModelParameters.phasesy_target[3] := 2.814228928151873;
stInitData.ModelParameters.phasesy_target[4] := 4.32353799667519;
stInitData.ModelParameters.phasesy_target[5] := 9.105215478795397;
stInitData.ModelParameters.phasesy_target[6] := 6.45749382748704;
stInitData.ModelParameters.phasesy_target[7] := -2.073824260704705;
stInitData.ModelParameters.phasesy_target[8] := -7.650625365765595;
stInitData.ModelParameters.phasesy_target[9] := 2.339476185381003;
stInitData.ModelParameters.phasesy_target[10] := 6.452393424316285;
stInitData.ModelParameters.phasesy_target[11] := -1.689364286355344;
stInitData.ModelParameters.phasesy_target[12] := -4.034195371452291;
stInitData.ModelParameters.phasesy_target[13] := 2.001331589298798;
stInitData.ModelParameters.phasesy_target[14] := 1.515933543855396;
stInitData.ModelParameters.phasesy_target[15] := 3.645294517897386;
stInitData.ModelParameters.phasesy_target[16] := 0.5515279517640805;
stInitData.ModelParameters.phasesy_target[17] := -0.07128093245878832;
stInitData.ModelParameters.phasesy_target[18] := -5.636407023395554;
stInitData.ModelParameters.phasesy_target[19] := -6.751800566422646;
stInitData.ModelParameters.phasesy_target[20] := 8.758470190795739;
stInitData.ModelParameters.phasesy_target[21] := 2.895252176566171;
stInitData.ModelParameters.phasesy_target[22] := 4.471560871325609;
stInitData.ModelParameters.phasesy_target[23] := -3.253689409343918;
stInitData.ModelParameters.phasesy_target[24] := -11.37771976330998;
stInitData.ModelParameters.phasesy_target[25] := 5.359774194580628;
stInitData.ModelParameters.phasesy_target[26] := 0.7392363080326961;
stInitData.ModelParameters.phasesy_target[27] := 4.427434833892008;
stInitData.ModelParameters.phasesy_target[28] := 12.24555683693308;
stInitData.ModelParameters.phasesy_target[29] := 4.938192454528604;
stInitData.ModelParameters.phasesy_target[30] := -8.164275301314767;
stInitData.ModelParameters.phasesy_target[31] := -2.428973204480333;
stInitData.ModelParameters.phasesy_target[32] := 0.2038225361798162;
stInitData.ModelParameters.phasesy_target[33] := -3.892901494998914;
stInitData.ModelParameters.phasesy_target[34] := 13.19207738739042;
stInitData.ModelParameters.phasesy_target[35] := -3.479174551435766;
stInitData.ModelParameters.phasesy_target[36] := -2.927185375361415;
stInitData.ModelParameters.phasesy_target[37] := -1.07284440266518;
stInitData.ModelParameters.phasesy_target[38] := 5.683447152525068;
stInitData.ModelParameters.phasesy_target[39] := -13.40647299389927;
stInitData.ModelParameters.phasesy_target[40] := -4.470062860893761;
stInitData.ModelParameters.phasesy_target[41] := -12.08214208794182;
stInitData.ModelParameters.phasesy_target[42] := 4.470357314800753;
stInitData.ModelParameters.phasesy_target[43] := -11.65116222216564;
stInitData.ModelParameters.phasesy_target[44] := 4.69916866043127;
stInitData.ModelParameters.phasesy_target[45] := 1.138234678416931;
stInitData.ModelParameters.phasesy_target[46] := 1.125825250134124;
stInitData.ModelParameters.phasesy_target[47] := 3.581561613121185;
stInitData.ModelParameters.phasesy_target[48] := -4.351822000667074;
stInitData.ModelParameters.phasesy_target[49] := -1.174920032929796;
stInitData.ModelParameters.phasesy_target[50] := 0.7515942483407694;
stInitData.ModelParameters.phasesy_target[51] := -9.623453417760389;
stInitData.ModelParameters.phasesy_target[52] := 2.895459428719547;
stInitData.ModelParameters.phasesy_target[53] := -5.982325255220389;
stInitData.ModelParameters.phasesy_target[54] := 0.07525689433432255;
stInitData.ModelParameters.phasesy_target[55] := -12.58825253483244;
stInitData.ModelParameters.phasesy_target[56] := 4.728794818011147;
stInitData.ModelParameters.phasesy_target[57] := -2.310500010252531;
stInitData.ModelParameters.phasesy_target[58] := -1.775141427594348;
stInitData.ModelParameters.phasesy_target[59] := -5.892907994877442;
stInitData.ModelParameters.phasesy_target[60] := 2.154910575317775;
stInitData.ModelParameters.phasesy_target[61] := -2.009151500716962;
stInitData.ModelParameters.phasesy_target[62] := 1.550326121117545;
stInitData.ModelParameters.phasesy_target[63] := 2.91517232446701;
stInitData.ModelParameters.phasesy_target[64] := 2.048514541205734;
stInitData.ModelParameters.phasesy_target[65] := -8.52681691758294;
stInitData.ModelParameters.phasesy_target[66] := -0.392716009279781;
stInitData.ModelParameters.phasesy_target[67] := 11.05232909291785;
stInitData.ModelParameters.phasesy_target[68] := 6.661621160806724;
stInitData.ModelParameters.phasesy_target[69] := -0.6449074706954264;
stInitData.ModelParameters.phasesy_target[70] := -6.663995288318766;
stInitData.ModelParameters.phasesy_target[71] := 1.938155591557062;
stInitData.ModelParameters.phasesy_target[72] := 9.698397677667341;
stInitData.ModelParameters.phasesy_target[73] := 14.03473796320933;
stInitData.ModelParameters.phasesy_target[74] := 7.030055920006444;
stInitData.ModelParameters.phasesy_target[75] := -0.7793874831010521;
stInitData.ModelParameters.phasesy_target[76] := 5.49895511361811;
stInitData.ModelParameters.phasesy_target[77] := -3.016009507925126;
stInitData.ModelParameters.phasesy_target[78] := 14.61837948033856;
stInitData.ModelParameters.phasesy_target[79] := -7.079852763538399;
stInitData.ModelParameters.phasesy_target[80] := -5.902535132569551;
stInitData.ModelParameters.phasesy_target[81] := 12.13522496987175;
stInitData.ModelParameters.phasesy_target[82] := -9.005566036138333;
stInitData.ModelParameters.phasesy_target[83] := 0.9394274314870444;
stInitData.ModelParameters.phasesy_target[84] := 3.154805328606508;
stInitData.ModelParameters.phasesy_target[85] := 0.1556288225160352;
stInitData.ModelParameters.phasesy_target[86] := -6.297353644953342;
stInitData.ModelParameters.phasesy_target[87] := 3.205776984484515;
stInitData.ModelParameters.phasesy_target[88] := 6.858396477582;
stInitData.ModelParameters.phasesy_target[89] := 2.293583740240707;
stInitData.ModelParameters.phasesy_target[90] := 7.006819645266965;
stInitData.ModelParameters.phasesy_target[91] := -2.375431679182152;
stInitData.ModelParameters.phasesy_target[92] := 5.052109130033248;
stInitData.ModelParameters.phasesy_target[93] := 3.138552360868532;
stInitData.ModelParameters.phasesy_target[94] := -4.263799659466268;
stInitData.ModelParameters.phasesy_target[95] := -2.723904418015559;
stInitData.ModelParameters.phasesy_target[96] := 2.703228531061528;
stInitData.ModelParameters.phasesy_target[97] := -0.05505587896275287;
stInitData.ModelParameters.phasesy_target[98] := -5.609522377682545;
stInitData.ModelParameters.phasesy_target[99] := -3.365819819714671;
stInitData.ModelParameters.phasesy_target[100] := 0.7593857263450322;
stInitData.ModelParameters.phasesy_target[101] := -4.152593855099633;
stInitData.ModelParameters.phasesy_target[102] := -2.648660152891155;
stInitData.ModelParameters.phasesy_target[103] := -2.595912162619209;
stInitData.ModelParameters.phasesy_target[104] := -3.474204571933332;
stInitData.ModelParameters.phasesy_target[105] := 0.2624215696204276;
stInitData.ModelParameters.phasesy_target[106] := 7.861845682457719;
stInitData.ModelParameters.phasesy_target[107] := -6.250862589118591;
stInitData.ModelParameters.phasesy_target[108] := -3.605220353567508;
stInitData.ModelParameters.phasesy_target[109] := -0.6334732298428778;
stInitData.ModelParameters.phasesy_target[110] := -0.0225958599468116;
stInitData.ModelParameters.phasesy_target[111] := 1.195264456311429;
stInitData.ModelParameters.phasesy_target[112] := 11.13994116767669;
stInitData.ModelParameters.phasesy_target[113] := -2.319670916476096;
stInitData.ModelParameters.phasesy_target[114] := 2.665809699694549;
stInitData.ModelParameters.phasesy_target[115] := 4.883288602907725;
stInitData.ModelParameters.phasesy_target[116] := 16.35338862577333;
stInitData.ModelParameters.phasesy_target[117] := -6.440192301685399;
stInitData.ModelParameters.phasesy_target[118] := 0.06521006642298283;
stInitData.ModelParameters.phasesy_target[119] := 1.975427544661816;
stInitData.ModelParameters.sampleTime := 0.001;
stInitData.ModelParameters.DiscreteDerivative_ICPrevScaled := 0;
stInitData.ModelParameters.DiscreteDerivative_ICPrevScal_e := 0;
stInitData.ModelParameters.DiscreteDerivative_ICPrevScal_m := 0;
stInitData.ModelParameters.DiscreteDerivative_ICPrevScal_h := 0;
stInitData.ModelParameters.DiscreteDerivative_ICPrevScal_c := 0;
stInitData.ModelParameters.DiscreteDerivative_ICPrevScal_g := 0;
stInitData.ModelParameters.DiscreteDerivative_ICPrevScal_d := 0;
stInitData.ModelParameters.DiscreteDerivative_ICPrevScal_i := 0;
stInitData.ModelParameters.DiscreteDerivative_ICPrevSca_hd := 0;
stInitData.ModelParameters.DiscreteDerivative_ICPrevScal_l := 0;
stInitData.ModelParameters.DiscreteDerivative_ICPrevScal_b := 0;
stInitData.ModelParameters.DiscreteDerivative_ICPrevSca_h3 := 0;
stInitData.ModelParameters.CompareToConstant_const := 0;
stInitData.ModelParameters.CompareToConstant_const_i := 201;
stInitData.ModelParameters.CompareToConstant_const_b := 0;
stInitData.ModelParameters.CompareToConstant_const_f := 201;
stInitData.ModelParameters.CompareToConstant_const_g := 0;
stInitData.ModelParameters.CompareToConstant_const_k := 4;
stInitData.ModelParameters.CompareToConstant_const_n := 4;
stInitData.ModelParameters.CompareToConstant1_const := 2.75;
stInitData.ModelParameters.CompareToConstant_const_j := 4;
stInitData.ModelParameters.CompareToConstant1_const_f := 2.75;
stInitData.ModelParameters.WrapToZero_Threshold := -1;
stInitData.ModelParameters.CompareToConstant_const_e := 0;
stInitData.ModelParameters.CompareToConstant_const_c := 0;
stInitData.ModelParameters.CompareToConstant_const_ew := 0;
stInitData.ModelParameters.CompareToConstant_const_if := 0;
stInitData.ModelParameters.ErrorHasOccurred_initial_condit := 0;
stInitData.ModelParameters.ErrorHasOccurred_initial_cond_l := 0;
stInitData.ModelParameters.ErrorHasOccurred_initial_con_ls := 0;
stInitData.ModelParameters.ErrorHasOccurred_initial_cond_c := 0;
stInitData.ModelParameters.CheckTrialIsRunning_initial_con := 0;
stInitData.ModelParameters.DetectRisePositive_vinit := 0;
stInitData.ModelParameters.DetectRisePositive1_vinit := 0;
stInitData.ModelParameters.DetectRisePositive_vinit_j := 0;
stInitData.ModelParameters.DetectRisePositive1_vinit_i := 0;
stInitData.ModelParameters.DetectRiseNonnegative_vinit := 0;
stInitData.ModelParameters.DetectIncrease_vinit := 0;
stInitData.ModelParameters.DetectRisePositive_vinit_h := 0;
stInitData.ModelParameters.DetectRisePositive1_vinit_o := 0;
stInitData.ModelParameters.DetectRisePositive_vinit_b := 0;
stInitData.ModelParameters.DetectRisePositive1_vinit_f := 0;
stInitData.ModelParameters.DetectChange_vinit := 0;
stInitData.ModelParameters.DetectChange_vinit_i := 0;
stInitData.ModelParameters.DetectChange_vinit_f := 0;
stInitData.ModelParameters.DetectChange_vinit_e := 0;
stInitData.ModelParameters.DetectIncrease_vinit_f := 0;
stInitData.ModelParameters.DetectRisePositive_vinit_k := 0;
stInitData.ModelParameters.DetectRisePositive1_vinit_b := 0;
stInitData.ModelParameters.Constant_Value := 1;
stInitData.ModelParameters.x_prev_InitialCondition := 0;
stInitData.ModelParameters.xdot_prev_InitialCondition := 0;
stInitData.ModelParameters.Constant_Value_j := 1;
stInitData.ModelParameters.x_prev_InitialCondition_g := 0;
stInitData.ModelParameters.xdot_prev_InitialCondition_f := 0;
stInitData.ModelParameters.JointTorqueDes_Nm_Y0[0] := 0;
stInitData.ModelParameters.JointTorqueDes_Nm_Y0[1] := 0;
stInitData.ModelParameters.Constant3_Value[0] := 0;
stInitData.ModelParameters.Constant3_Value[1] := 0;
stInitData.ModelParameters.JointTorqueDes_Nm_Y0_g[0] := 0;
stInitData.ModelParameters.JointTorqueDes_Nm_Y0_g[1] := 0;
stInitData.ModelParameters.Constant3_Value_f[0] := 0;
stInitData.ModelParameters.Constant3_Value_f[1] := 0;
stInitData.ModelParameters.JointTorqueDes_Nm_Y0_a[0] := 0;
stInitData.ModelParameters.JointTorqueDes_Nm_Y0_a[1] := 0;
stInitData.ModelParameters.Constant3_Value_l[0] := 0;
stInitData.ModelParameters.Constant3_Value_l[1] := 0;
stInitData.ModelParameters.JointTorqueDes_Nm_Y0_h[0] := 0;
stInitData.ModelParameters.JointTorqueDes_Nm_Y0_h[1] := 0;
stInitData.ModelParameters.Constant3_Value_o[0] := 0;
stInitData.ModelParameters.Constant3_Value_o[1] := 0;
stInitData.ModelParameters.Requestedstate_Value := 0;
stInitData.ModelParameters.CalibrateManually_Value := 0;
stInitData.ModelParameters.Memory_X0 := 0;
stInitData.ModelParameters.FreqHz_Value := 20;
stInitData.ModelParameters.UnitDelay_InitialCondition := 0;
stInitData.ModelParameters.TSamp_WtEt := 1000;
stInitData.ModelParameters.Butterworthfilter_InitialStates := 0;
stInitData.ModelParameters.Butterworthfilter_InitialDenomi := 0;
stInitData.ModelParameters.CalibrateManually_Value_p := 0;
stInitData.ModelParameters.FreqHz_Value_m := 20;
stInitData.ModelParameters.UnitDelay_InitialCondition_f := 0;
stInitData.ModelParameters.TSamp_WtEt_a := 1000;
stInitData.ModelParameters.Butterworthfilter_InitialStat_a := 0;
stInitData.ModelParameters.Butterworthfilter_InitialDeno_l := 0;
stInitData.ModelParameters.Constant2_Value := 0.05;
stInitData.ModelParameters.target3_Value[0] := 0;
stInitData.ModelParameters.target3_Value[1] := 0.25;
stInitData.ModelParameters.CalibrateManually_Value_c := 0;
stInitData.ModelParameters.Memory_X0_m := 0;
stInitData.ModelParameters.FreqHz_Value_f := 20;
stInitData.ModelParameters.UnitDelay_InitialCondition_j := 0;
stInitData.ModelParameters.TSamp_WtEt_p := 1000;
stInitData.ModelParameters.Butterworthfilter_InitialStat_m := 0;
stInitData.ModelParameters.Butterworthfilter_InitialDeno_p := 0;
stInitData.ModelParameters.CalibrateManually_Value_f := 0;
stInitData.ModelParameters.FreqHz_Value_j := 20;
stInitData.ModelParameters.UnitDelay_InitialCondition_a := 0;
stInitData.ModelParameters.TSamp_WtEt_b := 1000;
stInitData.ModelParameters.Butterworthfilter_InitialStat_j := 0;
stInitData.ModelParameters.Butterworthfilter_InitialDeno_i := 0;
stInitData.ModelParameters.Constant2_Value_a := 0.05;
stInitData.ModelParameters.target4_Value[0] := 0;
stInitData.ModelParameters.target4_Value[1] := 0.25;
stInitData.ModelParameters.EnableDrives_Value := 0;
stInitData.ModelParameters.UseActuator_Value := 1;
stInitData.ModelParameters.DisableDrives_Value := 0;
stInitData.ModelParameters.Constant_Value_l := 0;
stInitData.ModelParameters.TSamp_WtEt_f := 1000;
stInitData.ModelParameters.FreqHz_Value_mf := 100;
stInitData.ModelParameters.UnitDelay_InitialCondition_d := 0;
stInitData.ModelParameters.Constant_Value_m := 18.84955592153876;
stInitData.ModelParameters.AbsoluteMaximumTorque_Nm_Value := 8;
stInitData.ModelParameters.Bias_Bias := 0.5;
stInitData.ModelParameters.InhibitTime_s_Value := 2;
stInitData.ModelParameters.Memory1_1_X0 := 0;
stInitData.ModelParameters.Constant_Value_f := 0;
stInitData.ModelParameters.UseActuator_Value_h := 1;
stInitData.ModelParameters.Constant_Value_o := 0;
stInitData.ModelParameters.TSamp_WtEt_j := 1000;
stInitData.ModelParameters.FreqHz_Value_js := 100;
stInitData.ModelParameters.UnitDelay_InitialCondition_b := 0;
stInitData.ModelParameters.Constant_Value_c := 18.84955592153876;
stInitData.ModelParameters.AbsoluteMaximumTorque_Nm_Valu_k := 8;
stInitData.ModelParameters.Bias_Bias_j := 0.5;
stInitData.ModelParameters.InhibitTime_s_Value_f := 2;
stInitData.ModelParameters.Memory1_1_X0_h := 0;
stInitData.ModelParameters.TimePerState_ms_Value[0] := 50;
stInitData.ModelParameters.TimePerState_ms_Value[1] := 50;
stInitData.ModelParameters.TimePerState_ms_Value[2] := 150;
stInitData.ModelParameters.TimePerState_ms_Value[3] := 150;
stInitData.ModelParameters.SetModeOp_val_slx_Value := 10;
stInitData.ModelParameters.TorqueLimit_Value := 6;
stInitData.ModelParameters.virtualmass_Value := 0.5;
stInitData.ModelParameters.virtualdamping_Value := 0.05;
stInitData.ModelParameters.CalibrateForceSensors_Value := 0;
stInitData.ModelParameters.Constant_Value_b := 0;
stInitData.ModelParameters.KpConnection_Value := 0;
stInitData.ModelParameters.KdConnection_Value := 0;
stInitData.ModelParameters.TSamp_WtEt_k := 1000;
stInitData.ModelParameters.Butterworthfilter_InitialStat_o := 0;
stInitData.ModelParameters.Butterworthfilter_InitialDeno_h := 0;
stInitData.ModelParameters.TSamp_WtEt_kh := 1000;
stInitData.ModelParameters.Butterworthfilter_InitialSta_my := 0;
stInitData.ModelParameters.Butterworthfilter_InitialDeno_k := 0;
stInitData.ModelParameters.TSamp_WtEt_o := 1000;
stInitData.ModelParameters.Butterworthfilter_InitialStat_p := 0;
stInitData.ModelParameters.Butterworthfilter_InitialDeno_g := 0;
stInitData.ModelParameters.TSamp_WtEt_m := 1000;
stInitData.ModelParameters.Butterworthfilter_InitialStat_k := 0;
stInitData.ModelParameters.Butterworthfilter_InitialDen_hr := 0;
stInitData.ModelParameters.Merge1_InitialOutput[0] := 0;
stInitData.ModelParameters.Merge1_InitialOutput[1] := 0;
stInitData.ModelParameters.Kp_Gain := 1000;
stInitData.ModelParameters.Merge2_InitialOutput[0] := 0;
stInitData.ModelParameters.Merge2_InitialOutput[1] := 0;
stInitData.ModelParameters.Kd_Gain := 8;
stInitData.ModelParameters.Kd1_Gain := 0;
stInitData.ModelParameters.Kd2_Gain := 8;
stInitData.ModelParameters.Gain_Gain := 0;
stInitData.ModelParameters.TimePerState_ms_Value_n[0] := 50;
stInitData.ModelParameters.TimePerState_ms_Value_n[1] := 50;
stInitData.ModelParameters.TimePerState_ms_Value_n[2] := 150;
stInitData.ModelParameters.TimePerState_ms_Value_n[3] := 150;
stInitData.ModelParameters.SetModeOp_val_slx_Value_j := 10;
stInitData.ModelParameters.UseActuator_Value_f := 1;
stInitData.ModelParameters.Constant_Value_j1 := 0;
stInitData.ModelParameters.TSamp_WtEt_h := 1000;
stInitData.ModelParameters.FreqHz_Value_o := 100;
stInitData.ModelParameters.UnitDelay_InitialCondition_n := 0;
stInitData.ModelParameters.Constant_Value_jn := 18.84955592153876;
stInitData.ModelParameters.AbsoluteMaximumTorque_Nm_Valu_c := 8;
stInitData.ModelParameters.Bias_Bias_f := 0.5;
stInitData.ModelParameters.InhibitTime_s_Value_g := 2;
stInitData.ModelParameters.Memory1_1_X0_f := 0;
stInitData.ModelParameters.Constant_Value_jk := 0;
stInitData.ModelParameters.UseActuator_Value_l := 1;
stInitData.ModelParameters.Constant_Value_od := 0;
stInitData.ModelParameters.TSamp_WtEt_l := 1000;
stInitData.ModelParameters.FreqHz_Value_j5 := 100;
stInitData.ModelParameters.UnitDelay_InitialCondition_nf := 0;
stInitData.ModelParameters.Constant_Value_p := 18.84955592153876;
stInitData.ModelParameters.AbsoluteMaximumTorque_Nm_Valu_l := 8;
stInitData.ModelParameters.Bias_Bias_a := 0.5;
stInitData.ModelParameters.InhibitTime_s_Value_m := 2;
stInitData.ModelParameters.Memory1_1_X0_fk := 0;
stInitData.ModelParameters.TimePerState_ms_Value_d[0] := 50;
stInitData.ModelParameters.TimePerState_ms_Value_d[1] := 50;
stInitData.ModelParameters.TimePerState_ms_Value_d[2] := 150;
stInitData.ModelParameters.TimePerState_ms_Value_d[3] := 150;
stInitData.ModelParameters.SetModeOp_val_slx_Value_n := 10;
stInitData.ModelParameters.TorqueLimit_Value_m := 4;
stInitData.ModelParameters.ExpTrialRandom1_Value[0] := 0;
stInitData.ModelParameters.ExpTrialRandom1_Value[1] := 0;
stInitData.ModelParameters.ExpTrialRandom2_Value[0] := 0;
stInitData.ModelParameters.ExpTrialRandom2_Value[1] := 0;
stInitData.ModelParameters.Merge1_InitialOutput_e[0] := 0;
stInitData.ModelParameters.Merge1_InitialOutput_e[1] := 0;
stInitData.ModelParameters.Kp_Gain_m := 1000;
stInitData.ModelParameters.Merge2_InitialOutput_k[0] := 0;
stInitData.ModelParameters.Merge2_InitialOutput_k[1] := 0;
stInitData.ModelParameters.Kd_Gain_i := 8;
stInitData.ModelParameters.Kd1_Gain_n := 0;
stInitData.ModelParameters.Kd2_Gain_k := 8;
stInitData.ModelParameters.Gain_Gain_h := 0;
stInitData.ModelParameters.TimePerState_ms_Value_e[0] := 50;
stInitData.ModelParameters.TimePerState_ms_Value_e[1] := 50;
stInitData.ModelParameters.TimePerState_ms_Value_e[2] := 150;
stInitData.ModelParameters.TimePerState_ms_Value_e[3] := 150;
stInitData.ModelParameters.SetModeOp_val_slx_Value_p := 10;
stInitData.ModelParameters.One_Value := 1;
stInitData.ModelParameters.ExpStartTrial_Value := 0;
stInitData.ModelParameters.Constant_Value_n := 0;
stInitData.ModelParameters.ExpTrialIntroDuration_Value := 5;
stInitData.ModelParameters.ExpTrialDuration_Value := 30;
stInitData.ModelParameters.RateLimiter_RisingLim := 0.0003333333333333333;
stInitData.ModelParameters.RateLimiter_FallingLim := -0.00025;
stInitData.ModelParameters.RateLimiter_IC := 0;
stInitData.ModelParameters.Saturation_UpperSat := 1;
stInitData.ModelParameters.Saturation_LowerSat := 0;
stInitData.ModelParameters.Gain1_Gain := 6.283185307179586;
stInitData.ModelParameters.Gain2_Gain := 0.1591549430918953;
stInitData.ModelParameters.Saturation_UpperSat_h := 1;
stInitData.ModelParameters.Saturation_LowerSat_f := 0;
stInitData.ModelParameters.One_Value_h := 1;
stInitData.ModelParameters.Saturation_UpperSat_o := 1;
stInitData.ModelParameters.Saturation_LowerSat_fc := 0;
stInitData.ModelParameters.rotation_Value := 1.047197551196598;
stInitData.ModelParameters.Merge3_InitialOutput[0] := 0;
stInitData.ModelParameters.Merge3_InitialOutput[1] := 0;
stInitData.ModelParameters.Memory1_10_X0 := 0;
stInitData.ModelParameters.Memory1_11_X0 := 0;
stInitData.ModelParameters.Memory1_2_X0 := 0;
stInitData.ModelParameters.Memory1_3_X0 := 0;
stInitData.ModelParameters.Memory1_4_X0 := 0;
stInitData.ModelParameters.Memory1_5_X0 := 0;
stInitData.ModelParameters.Memory1_6_X0 := 0;
stInitData.ModelParameters.Memory1_7_X0 := 0;
stInitData.ModelParameters.Memory1_8_X0 := 0;
stInitData.ModelParameters.Memory1_9_X0 := 0;
stInitData.ModelParameters.Memory1_10_X0_h := 0;
stInitData.ModelParameters.Memory1_11_X0_h := 0;
stInitData.ModelParameters.Memory1_2_X0_h := 0;
stInitData.ModelParameters.Memory1_3_X0_h := 0;
stInitData.ModelParameters.Memory1_4_X0_h := 0;
stInitData.ModelParameters.Memory1_5_X0_h := 0;
stInitData.ModelParameters.Memory1_6_X0_h := 0;
stInitData.ModelParameters.Memory1_7_X0_h := 0;
stInitData.ModelParameters.Memory1_8_X0_h := 0;
stInitData.ModelParameters.Memory1_9_X0_h := 0;
stInitData.ModelParameters.Merge3_InitialOutput_m[0] := 0;
stInitData.ModelParameters.Merge3_InitialOutput_m[1] := 0;
stInitData.ModelParameters.Memory1_10_X0_f := 0;
stInitData.ModelParameters.Memory1_11_X0_f := 0;
stInitData.ModelParameters.Memory1_2_X0_f := 0;
stInitData.ModelParameters.Memory1_3_X0_f := 0;
stInitData.ModelParameters.Memory1_4_X0_f := 0;
stInitData.ModelParameters.Memory1_5_X0_f := 0;
stInitData.ModelParameters.Memory1_6_X0_f := 0;
stInitData.ModelParameters.Memory1_7_X0_f := 0;
stInitData.ModelParameters.Memory1_8_X0_f := 0;
stInitData.ModelParameters.Memory1_9_X0_f := 0;
stInitData.ModelParameters.Memory1_10_X0_fk := 0;
stInitData.ModelParameters.Memory1_11_X0_fk := 0;
stInitData.ModelParameters.Memory1_2_X0_fk := 0;
stInitData.ModelParameters.Memory1_3_X0_fk := 0;
stInitData.ModelParameters.Memory1_4_X0_fk := 0;
stInitData.ModelParameters.Memory1_5_X0_fk := 0;
stInitData.ModelParameters.Memory1_6_X0_fk := 0;
stInitData.ModelParameters.Memory1_7_X0_fk := 0;
stInitData.ModelParameters.Memory1_8_X0_fk := 0;
stInitData.ModelParameters.Memory1_9_X0_fk := 0;
stInitData.ModelParameters.Recorddata1yes0no_Value := 0;
stInitData.ModelParameters.Gain_Gain_e := 1;
stInitData.ModelParameters.ExpTrialRandom3_Value[0] := 0;
stInitData.ModelParameters.ExpTrialRandom3_Value[1] := 0;
stInitData.ModelParameters.ExpTrialRandom_Value := 1;
stInitData.ModelParameters.ExpTrialRandom4_Value[0] := 0;
stInitData.ModelParameters.ExpTrialRandom4_Value[1] := 0;
stInitData.ModelParameters.ExpCondition_Value := 0;
stInitData.ModelParameters.ExpTrialNumber1_Value := 1;
stInitData.ModelParameters.FixPtConstant_Value := 1;
stInitData.ModelParameters.Output_InitialCondition := 0;
stInitData.ModelParameters.Constant_Value_g := 0;
stInitData.ModelParameters.ManualSwitch_CurrentSetting := 0;
stInitData.ModelParameters.ManualSwitch_CurrentSetting_m := 0;
stInitData.ModelParameters.ManualSwitch_CurrentSetting_h := 0;
stInitData.ModelParameters.ManualSwitch_CurrentSetting_j := 0;
stInitData.ModelParameters.Memory1_X0 := 0;
stInitData.ModelParameters.PreventAlgebraicLoop_X0 := 0;
stInitData.ModelParameters.PreventAlgebraicLoop_X0_m := 0;
stInitData.ModelParameters.AvoidAlgebraicLoop_X0 := 0;
stInitData.ModelParameters.AvoidAlgebraicLoop_X0_k := 0;
stInitData.ModelParameters.PreventAlgebraicLoop_X0_h := 0;
stInitData.ModelParameters.PreventAlgebraicLoop_X0_o := 0;
stInitData.ModelParameters.AvoidAlgebraicLoop_X0_l := 0;
stInitData.ModelParameters.AvoidAlgebraicLoop_X0_b := 0;
stInitData.ModelParameters.Constant_Value_h := 0;
stInitData.ModelParameters.Memory_X0_n := 0;
stInitData.ModelParameters.Constant_Value_lx := 0;
stInitData.ModelParameters.Constant_Value_hx := 0;
stInitData.ModelParameters.Logic_table[0] := 0;
stInitData.ModelParameters.Logic_table[1] := 1;
stInitData.ModelParameters.Logic_table[2] := 0;
stInitData.ModelParameters.Logic_table[3] := 0;
stInitData.ModelParameters.Logic_table[4] := 1;
stInitData.ModelParameters.Logic_table[5] := 1;
stInitData.ModelParameters.Logic_table[6] := 0;
stInitData.ModelParameters.Logic_table[7] := 0;
stInitData.ModelParameters.Logic_table[8] := 1;
stInitData.ModelParameters.Logic_table[9] := 0;
stInitData.ModelParameters.Logic_table[10] := 1;
stInitData.ModelParameters.Logic_table[11] := 1;
stInitData.ModelParameters.Logic_table[12] := 0;
stInitData.ModelParameters.Logic_table[13] := 0;
stInitData.ModelParameters.Logic_table[14] := 0;
stInitData.ModelParameters.Logic_table[15] := 0;
stInitData.ModelParameters.Memory1_X0_p := 0;
stInitData.ModelParameters.Constant_Value_gf := 0;
stInitData.ModelParameters.Memory_X0_k := 0;
stInitData.ModelParameters.Constant_Value_cq := 0;
stInitData.ModelParameters.Constant_Value_i := 0;
stInitData.ModelParameters.Logic_table_h[0] := 0;
stInitData.ModelParameters.Logic_table_h[1] := 1;
stInitData.ModelParameters.Logic_table_h[2] := 0;
stInitData.ModelParameters.Logic_table_h[3] := 0;
stInitData.ModelParameters.Logic_table_h[4] := 1;
stInitData.ModelParameters.Logic_table_h[5] := 1;
stInitData.ModelParameters.Logic_table_h[6] := 0;
stInitData.ModelParameters.Logic_table_h[7] := 0;
stInitData.ModelParameters.Logic_table_h[8] := 1;
stInitData.ModelParameters.Logic_table_h[9] := 0;
stInitData.ModelParameters.Logic_table_h[10] := 1;
stInitData.ModelParameters.Logic_table_h[11] := 1;
stInitData.ModelParameters.Logic_table_h[12] := 0;
stInitData.ModelParameters.Logic_table_h[13] := 0;
stInitData.ModelParameters.Logic_table_h[14] := 0;
stInitData.ModelParameters.Logic_table_h[15] := 0;
stInitData.ModelParameters.Connected_Value := 0;
stInitData.ModelParameters.Memory1_X0_pr := 0;
stInitData.ModelParameters.Constant_Value_cx := 0;
stInitData.ModelParameters.Memory_X0_nw := 0;
stInitData.ModelParameters.Constant_Value_k := 0;
stInitData.ModelParameters.Constant_Value_oq := 0;
stInitData.ModelParameters.Logic_table_f[0] := 0;
stInitData.ModelParameters.Logic_table_f[1] := 1;
stInitData.ModelParameters.Logic_table_f[2] := 0;
stInitData.ModelParameters.Logic_table_f[3] := 0;
stInitData.ModelParameters.Logic_table_f[4] := 1;
stInitData.ModelParameters.Logic_table_f[5] := 1;
stInitData.ModelParameters.Logic_table_f[6] := 0;
stInitData.ModelParameters.Logic_table_f[7] := 0;
stInitData.ModelParameters.Logic_table_f[8] := 1;
stInitData.ModelParameters.Logic_table_f[9] := 0;
stInitData.ModelParameters.Logic_table_f[10] := 1;
stInitData.ModelParameters.Logic_table_f[11] := 1;
stInitData.ModelParameters.Logic_table_f[12] := 0;
stInitData.ModelParameters.Logic_table_f[13] := 0;
stInitData.ModelParameters.Logic_table_f[14] := 0;
stInitData.ModelParameters.Logic_table_f[15] := 0;
stInitData.ModelParameters.Memory1_X0_i := 0;
stInitData.ModelParameters.Constant_Value_ky := 0;
stInitData.ModelParameters.Memory_X0_p := 0;
stInitData.ModelParameters.Constant_Value_kl := 0;
stInitData.ModelParameters.Constant_Value_m5 := 0;
stInitData.ModelParameters.Logic_table_i[0] := 0;
stInitData.ModelParameters.Logic_table_i[1] := 1;
stInitData.ModelParameters.Logic_table_i[2] := 0;
stInitData.ModelParameters.Logic_table_i[3] := 0;
stInitData.ModelParameters.Logic_table_i[4] := 1;
stInitData.ModelParameters.Logic_table_i[5] := 1;
stInitData.ModelParameters.Logic_table_i[6] := 0;
stInitData.ModelParameters.Logic_table_i[7] := 0;
stInitData.ModelParameters.Logic_table_i[8] := 1;
stInitData.ModelParameters.Logic_table_i[9] := 0;
stInitData.ModelParameters.Logic_table_i[10] := 1;
stInitData.ModelParameters.Logic_table_i[11] := 1;
stInitData.ModelParameters.Logic_table_i[12] := 0;
stInitData.ModelParameters.Logic_table_i[13] := 0;
stInitData.ModelParameters.Logic_table_i[14] := 0;
stInitData.ModelParameters.Logic_table_i[15] := 0;
stInitData.ModelParameters.Memory_X0_i := 0;
stInitData.ModelParameters.Memory_X0_h := 0;
stInitData.ModelParameters.Memory_X0_pu := 0;
stInitData.ModelParameters.Memory_X0_j := 0;
stInitData.ModelParameters.Memory_X0_l := 0;
stInitData.ModelParameters.Constant_Value_hh := 0;
stInitData.ModelParameters.Logic_table_f1[0] := 0;
stInitData.ModelParameters.Logic_table_f1[1] := 1;
stInitData.ModelParameters.Logic_table_f1[2] := 0;
stInitData.ModelParameters.Logic_table_f1[3] := 0;
stInitData.ModelParameters.Logic_table_f1[4] := 1;
stInitData.ModelParameters.Logic_table_f1[5] := 1;
stInitData.ModelParameters.Logic_table_f1[6] := 0;
stInitData.ModelParameters.Logic_table_f1[7] := 0;
stInitData.ModelParameters.Logic_table_f1[8] := 1;
stInitData.ModelParameters.Logic_table_f1[9] := 0;
stInitData.ModelParameters.Logic_table_f1[10] := 1;
stInitData.ModelParameters.Logic_table_f1[11] := 1;
stInitData.ModelParameters.Logic_table_f1[12] := 0;
stInitData.ModelParameters.Logic_table_f1[13] := 0;
stInitData.ModelParameters.Logic_table_f1[14] := 0;
stInitData.ModelParameters.Logic_table_f1[15] := 0;
stInitData.ModelParameters.LatchRising_d.Out_Y0 := 0;
stInitData.ModelParameters.LatchRising_m.Out_Y0 := 0;
stInitData.ModelParameters.run_c.x_ref_Y0[0] := 0;
stInitData.ModelParameters.run_c.x_ref_Y0[1] := 0;
stInitData.ModelParameters.run_c.xdot_ref_Y0[0] := 0;
stInitData.ModelParameters.run_c.xdot_ref_Y0[1] := 0;
stInitData.ModelParameters.run_c.xddot_ref_Y0[0] := 0;
stInitData.ModelParameters.run_c.xddot_ref_Y0[1] := 0;
stInitData.ModelParameters.athome_g.WrapToZero_Threshold := -1;
stInitData.ModelParameters.athome_g.Memory1_X0 := 0;
stInitData.ModelParameters.athome_g.x_ref_Y0[0] := 0;
stInitData.ModelParameters.athome_g.x_ref_Y0[1] := 0;
stInitData.ModelParameters.athome_g.xdot_ref_Y0[0] := 0;
stInitData.ModelParameters.athome_g.xdot_ref_Y0[1] := 0;
stInitData.ModelParameters.athome_g.xddot_ref_Y0[0] := 0;
stInitData.ModelParameters.athome_g.xddot_ref_Y0[1] := 0;
stInitData.ModelParameters.athome_g.Constant_Value := 1;
stInitData.ModelParameters.athome_g.Constant2_Value[0] := 0;
stInitData.ModelParameters.athome_g.Constant2_Value[1] := 0;
stInitData.ModelParameters.athome_g.Constant4_Value[0] := 0;
stInitData.ModelParameters.athome_g.Constant4_Value[1] := 0;
stInitData.ModelParameters.athome_g.FixPtConstant_Value := 1;
stInitData.ModelParameters.athome_g.Output_InitialCondition := 0;
stInitData.ModelParameters.athome_g.Constant_Value_h := 0;
stInitData.ModelParameters.athome_g.Switch_Threshold := 1;
stInitData.ModelParameters.homingactive_d.x_ref_Y0[0] := 0;
stInitData.ModelParameters.homingactive_d.x_ref_Y0[1] := 0;
stInitData.ModelParameters.homingactive_d.xdot_ref_Y0[0] := 0;
stInitData.ModelParameters.homingactive_d.xdot_ref_Y0[1] := 0;
stInitData.ModelParameters.homingactive_d.xddot_ref_Y0[0] := 0;
stInitData.ModelParameters.homingactive_d.xddot_ref_Y0[1] := 0;
stInitData.ModelParameters.homingactive_d.Constant1_Value := 1;
stInitData.ModelParameters.homingactive_d.One_Value := 1;
stInitData.ModelParameters.homingactive_d.RateLimiter_RisingLim := 0.0001;
stInitData.ModelParameters.homingactive_d.RateLimiter_FallingLim := -0.0002;
stInitData.ModelParameters.homingactive_d.RateLimiter_IC := 0;
stInitData.ModelParameters.homingactive_d.Saturation_UpperSat := 1;
stInitData.ModelParameters.homingactive_d.Saturation_LowerSat := 0;
stInitData.ModelParameters.homingactive_d.Gain1_Gain := 6.283185307179586;
stInitData.ModelParameters.homingactive_d.Gain2_Gain := 0.1591549430918953;
stInitData.ModelParameters.homingactive_d.Saturation_UpperSat_h := 1;
stInitData.ModelParameters.homingactive_d.Saturation_LowerSat_d := 0;
stInitData.ModelParameters.homingactive_d.Constant2_Value[0] := 0;
stInitData.ModelParameters.homingactive_d.Constant2_Value[1] := 0;
stInitData.ModelParameters.homingactive_d.Constant4_Value[0] := 0;
stInitData.ModelParameters.homingactive_d.Constant4_Value[1] := 0;
stInitData.ModelParameters.LatchRising_c.Out_Y0 := 0;
stInitData.ModelParameters.LatchRising_b.Out_Y0 := 0;
stInitData.ModelParameters.run.x_ref_Y0[0] := 0;
stInitData.ModelParameters.run.x_ref_Y0[1] := 0;
stInitData.ModelParameters.run.xdot_ref_Y0[0] := 0;
stInitData.ModelParameters.run.xdot_ref_Y0[1] := 0;
stInitData.ModelParameters.run.xddot_ref_Y0[0] := 0;
stInitData.ModelParameters.run.xddot_ref_Y0[1] := 0;
stInitData.ModelParameters.athome.WrapToZero_Threshold := -1;
stInitData.ModelParameters.athome.Memory1_X0 := 0;
stInitData.ModelParameters.athome.x_ref_Y0[0] := 0;
stInitData.ModelParameters.athome.x_ref_Y0[1] := 0;
stInitData.ModelParameters.athome.xdot_ref_Y0[0] := 0;
stInitData.ModelParameters.athome.xdot_ref_Y0[1] := 0;
stInitData.ModelParameters.athome.xddot_ref_Y0[0] := 0;
stInitData.ModelParameters.athome.xddot_ref_Y0[1] := 0;
stInitData.ModelParameters.athome.Constant_Value := 1;
stInitData.ModelParameters.athome.Constant2_Value[0] := 0;
stInitData.ModelParameters.athome.Constant2_Value[1] := 0;
stInitData.ModelParameters.athome.Constant4_Value[0] := 0;
stInitData.ModelParameters.athome.Constant4_Value[1] := 0;
stInitData.ModelParameters.athome.FixPtConstant_Value := 1;
stInitData.ModelParameters.athome.Output_InitialCondition := 0;
stInitData.ModelParameters.athome.Constant_Value_h := 0;
stInitData.ModelParameters.athome.Switch_Threshold := 1;
stInitData.ModelParameters.homingactive.x_ref_Y0[0] := 0;
stInitData.ModelParameters.homingactive.x_ref_Y0[1] := 0;
stInitData.ModelParameters.homingactive.xdot_ref_Y0[0] := 0;
stInitData.ModelParameters.homingactive.xdot_ref_Y0[1] := 0;
stInitData.ModelParameters.homingactive.xddot_ref_Y0[0] := 0;
stInitData.ModelParameters.homingactive.xddot_ref_Y0[1] := 0;
stInitData.ModelParameters.homingactive.Constant1_Value := 1;
stInitData.ModelParameters.homingactive.One_Value := 1;
stInitData.ModelParameters.homingactive.RateLimiter_RisingLim := 0.0001;
stInitData.ModelParameters.homingactive.RateLimiter_FallingLim := -0.0002;
stInitData.ModelParameters.homingactive.RateLimiter_IC := 0;
stInitData.ModelParameters.homingactive.Saturation_UpperSat := 1;
stInitData.ModelParameters.homingactive.Saturation_LowerSat := 0;
stInitData.ModelParameters.homingactive.Gain1_Gain := 6.283185307179586;
stInitData.ModelParameters.homingactive.Gain2_Gain := 0.1591549430918953;
stInitData.ModelParameters.homingactive.Saturation_UpperSat_h := 1;
stInitData.ModelParameters.homingactive.Saturation_LowerSat_d := 0;
stInitData.ModelParameters.homingactive.Constant2_Value[0] := 0;
stInitData.ModelParameters.homingactive.Constant2_Value[1] := 0;
stInitData.ModelParameters.homingactive.Constant4_Value[0] := 0;
stInitData.ModelParameters.homingactive.Constant4_Value[1] := 0;
stInitData.ModelParameters.HoldFirstSampleOnEnable_e.WrapToZero_Threshold := -1;
stInitData.ModelParameters.HoldFirstSampleOnEnable_e.Memory1_X0 := 0;
stInitData.ModelParameters.HoldFirstSampleOnEnable_e.Output_InitialCondition := 0;
stInitData.ModelParameters.HoldFirstSampleOnEnable_e.Switch_Threshold := 1;
stInitData.ModelParameters.HoldFirstSampleOnEnable_e.FixPtConstant_Value := 1;
stInitData.ModelParameters.HoldFirstSampleOnEnable_e.Constant_Value := 0;
stInitData.ModelParameters.HoldFirstSampleOnEnable.WrapToZero_Threshold := -1;
stInitData.ModelParameters.HoldFirstSampleOnEnable.Memory1_X0 := 0;
stInitData.ModelParameters.HoldFirstSampleOnEnable.Output_InitialCondition := 0;
stInitData.ModelParameters.HoldFirstSampleOnEnable.Switch_Threshold := 1;
stInitData.ModelParameters.HoldFirstSampleOnEnable.FixPtConstant_Value := 1;
stInitData.ModelParameters.HoldFirstSampleOnEnable.Constant_Value := 0;
stInitData.ContextInfoArr_0_TaskOidHdr.indexGroup := 0;
stInitData.ContextInfoArr_0_TaskOidHdr.indexOffset := 16#03002060;
stInitData.ContextInfoArr_0_TaskOidHdr.cbData := SIZEOF(stInitData.ContextInfoArr_0_TaskOid);
stInitData.ContextInfoArr_0_TaskPriorityHdr.indexGroup := 0;
stInitData.ContextInfoArr_0_TaskPriorityHdr.indexOffset := 16#03002070;
stInitData.ContextInfoArr_0_TaskPriorityHdr.cbData := SIZEOF(stInitData.ContextInfoArr_0_TaskPriority);
stInitData.ContextInfoArr_0_TaskCycleTimeNsHdr.indexGroup := 0;
stInitData.ContextInfoArr_0_TaskCycleTimeNsHdr.indexOffset := 16#03002080;
stInitData.ContextInfoArr_0_TaskCycleTimeNsHdr.cbData := SIZEOF(stInitData.ContextInfoArr_0_TaskCycleTimeNs);
stInitData.ContextInfoArr_0_TaskPortHdr.indexGroup := 0;
stInitData.ContextInfoArr_0_TaskPortHdr.indexOffset := 16#03002090;
stInitData.ContextInfoArr_0_TaskPortHdr.cbData := SIZEOF(stInitData.ContextInfoArr_0_TaskPort);
stInitData.ContextInfoArr_0_TaskSortOrderHdr.indexGroup := 0;
stInitData.ContextInfoArr_0_TaskSortOrderHdr.indexOffset := 16#030020b0;
stInitData.ContextInfoArr_0_TaskSortOrderHdr.cbData := SIZEOF(stInitData.ContextInfoArr_0_TaskSortOrder);
stInitData.Header.cbData := SIZEOF(stInitData)-SIZEOF(stInitData.Header);
stInitData.Header.uiElmCnt := 12;


// set pointer to InitData structure
SetInitDataInfo(ADR(stInitData));

// set DataArea information
SetDataAreaInfo(ADR(arrDataAreas),2);
arrDataAreas[1].nDataAreaId := 0;
arrDataAreas[1].nSize := SIZEOF(stInput);
arrDataAreas[1].pPlcVar := ADR(stInput);
arrDataAreas[1].pModuleProcImg := 0;
arrDataAreas[1].eDataAreaType := E_TcMatSimDataAreaType.InputDst;
arrDataAreas[2].nDataAreaId := 1;
arrDataAreas[2].nSize := SIZEOF(stOutput);
arrDataAreas[2].pPlcVar := ADR(stOutput);
arrDataAreas[2].pModuleProcImg := 0;
arrDataAreas[2].eDataAreaType := E_TcMatSimDataAreaType.OutputSrc;


// initialize basic interface pointers and return
FB_init := SUCCEEDED(Init(oid));
                  
                
END_METHOD

METHOD Execute : HRESULT
                  
IF (SUCCEEDED(hResult)) THEN
  hResult := VerifyParameters();
END_IF

	// update DataArea information
SetDataAreaInfo(ADR(arrDataAreas),2);
	
	// call base method
Execute := SUPER^.Execute();
                  
                
END_METHOD

{attribute 'object_name' := 'VerifyParameters'}
METHOD VerifyParameters : HRESULT
  VAR
    moduleCallByParam : TctModuleCallByType;
  END_VAR
                  
IF (bParametersVerified) THEN
  VerifyParameters := Tc2_System.E_HRESULTAdsErr.HRESULT_ADS_NOERROR;
ELSE
  VerifyParameters := GetObjPara(stInitData.CallByHdr.indexOffset,SIZEOF(moduleCallByParam),ADR(moduleCallByParam));
  
  // check the "CallBy" parameter to be set to "Module"
  IF (SUCCEEDED(VerifyParameters) AND (moduleCallByParam <> TctModuleCallByType.Module)) THEN
      VerifyParameters := Tc2_System.E_HRESULTAdsErr.INVALIDPARM;
  END_IF
  
  // set the parameters verified flag
  bParametersVerified := SUCCEEDED(VerifyParameters);
END_IF
                  
                
END_METHOD

PROPERTY InitData : ST_ModelBROSMattia_InitData
GET
                    InitData := stInitData;
                  
END_GET
SET
                    stInitData := InitData;
                  
END_SET
END_PROPERTY
END_FUNCTION_BLOCK
